METHOD BrakeStatus 								: REFERENCE TO Tc2_MC2.ST_McOutputs
VAR_INPUT
	bExecute									: BOOL;
END_VAR
VAR_INST
	{attribute 'hide'}
	fbRead										: Tc2_EtherCAT.FB_CoERead_ByDriveRef;
	{attribute 'hide'}
	ftRead										: F_TRIG;
	{attribute 'hide'}
	nData										: BYTE;
END_VAR
VAR
	Out											: Tc2_MC2.ST_McOutputs;
END_VAR
fbRead			(	stDriveRef				:= _stDriveRef, 
					nIndex					:= 16#3001 + (_stDriveRef.nDriveNo * 16#400), 
					nSubIndex				:= 16#07, 
					pDstBuf					:= ADR(nData), 
					cbBufLen				:= SIZEOF(nData), 
					bExecute				:= bExecute,
					bBusy					=> Out.Busy, 
					bError					=> Out.Error, 
					iAdsErrId				=> , 
					iCANopenErrId			=> );

IF Out.Error THEN
	Out.ErrorID								:= fbRead.iAdsErrId + fbRead.iCANopenErrId;
END_IF
					
ftRead(CLK:= Out.Busy, Q=> );
IF ftRead.Q THEN
	Out.Done								:= NOT Out.Error;
	bHoldingBrakeUnlocked					:= nData.0;
	bHoldingBrakeLocked						:= NOT nData.0;
END_IF

BrakeStatus									REF= Out;
END_METHOD

METHOD DeletePositionOffset 					: REFERENCE TO Tc2_MC2.ST_McOutputs
VAR_INPUT
	bExecute									: BOOL;
	eFeedback									: Tc2_MC2_Drive.E_PositionOffsetFeedback;
	eMemory										: Tc2_MC2_Drive.E_PositionOffsetMemory;
END_VAR
IF bExecute THEN
	DeletePositionOffsetEx(	eFeedback			:= eFeedback, 
							eMemory				:= eMemory);
ELSE
	DeletePositionOffsetClear();
END_IF

DeletePositionOffset							REF= pDeletePosOffs;
END_METHOD

METHOD DeletePositionOffsetClear 				: BOOL
VAR
	{attribute 'hide'}
	Out											: ST_McOutputs;
END_VAR
VAR_INST
	{attribute 'hide'}
	ftBusy										: F_TRIG;
END_VAR
fbDeletePositionOffset(	Axis					:= Axis, 
						Execute					:= FALSE, 
						Feedback				:= , 
						Memory					:= , 
						Busy					=> Out.Busy, 
						Error					=> Out.Error, 
						ErrorID					=> Out.ErrorID);

ftBusy(CLK:= Out.Busy, Q=> );						
IF ftBusy.Q THEN
	Out.Done									:= NOT Out.Error;
END_IF

pDeletePosOffs									REF= Out;

DeletePositionOffsetClear						:= TRUE;
END_METHOD

METHOD DeletePositionOffsetEncoder 				: REFERENCE TO Tc2_MC2.ST_McOutputs
VAR_INPUT
	bExecute									: BOOL;
END_VAR
DeletePositionOffset(	bExecute				:= bExecute,
						eFeedback				:= Tc2_MC2_Drive.E_PositionOffsetFeedback.ePositionOffsetFeedback1, 
						eMemory					:= Tc2_MC2_Drive.E_PositionOffsetMemory.ePositionOffsetMemory_Encoder);

DeletePositionOffsetEncoder						REF= pDeletePosOffs;
END_METHOD

METHOD DeletePositionOffsetEx 					: BOOL
VAR_INPUT
	eFeedback									: Tc2_MC2_Drive.E_PositionOffsetFeedback;
	eMemory										: Tc2_MC2_Drive.E_PositionOffsetMemory;
END_VAR
VAR
	{attribute 'hide'}
	Out											: ST_McOutputs;
END_VAR
fbDeletePositionOffset(	Axis					:= Axis, 
						Execute					:= TRUE, 
						Feedback				:= eFeedback, 
						Memory					:= eMemory, 
						Busy					=> Out.Busy, 
						Error					=> Out.Error, 
						ErrorID					=> Out.ErrorID);
						
Out.Done										:= NOT Out.Error AND NOT Out.Busy;
pDeletePosOffs									REF= Out;

DeletePositionOffsetEx							:= TRUE;
END_METHOD

METHOD FB_Init 									: BOOL
VAR_INPUT
	bInitRetains 								: BOOL; // if TRUE, the retain variables are initialized (warm start / cold start)
	bInCopyCode 								: BOOL;  // if TRUE, the instance afterwards gets moved into the copy code (online change)
END_VAR
pDeletePosOffs									REF= _stDeletePosOffs;
pSetPosOffs										REF= _stSetPosOffs;
pDriveAddress									REF= _stDriveAddress;
pDriveRef										REF= _stDriveRef;
END_METHOD

{attribute 'monitoring' := 'variable'}
PROPERTY fTorqueLimit 					: LREAL
GET
fTorqueLimit									:= nBipolarTorqueLimitValue/10.0;
END_GET
SET
VAR CONSTANT
	rTorqueLimitLow								: REAL 		:= 0.01;				// Low limit used for bipolar torque limit value
	rTorqueLimitHigh							: REAL		:= 500.0;				// High limit used for bipolar torque limit value
END_VAR
IF fTorqueLimit < rTorqueLimitLow OR fTorqueLimit > rTorqueLimitHigh THEN
	nBipolarTorqueLimitValue 					:= LREAL_TO_UINT(rTorqueLimitHigh)*10;
ELSE
	nBipolarTorqueLimitValue 					:= LREAL_TO_UINT(fTorqueLimit)*10;
END_IF
END_SET
END_PROPERTY

METHOD PRIVATE GetDriveRef 						: REFERENCE TO Tc2_MC2.ST_McOutputs
VAR_INPUT
	bExecute									: BOOL;
END_VAR
VAR_INST
	{attribute 'hide'}
	fbGetDriveRef								: FB_GetDriveRef;
	{attribute 'hide'}
	ftRead										: F_TRIG;
END_VAR
VAR
	{attribute 'hide'}
	Out											: Tc2_MC2.ST_McOutputs;
END_VAR
fbGetDriveRef(	bExecute						:= bExecute, 
				bBusy							=> Out.Busy, 
				bError							=> Out.Error, 
				udiErrorID						=> Out.ErrorID, 
				stDriveRef						=> _stDriveRef, 
				Axis							:= Axis);
				
ftRead(CLK:= Out.Busy, Q=> );
IF ftRead.Q THEN
	Out.Done									:= NOT Out.Error;
END_IF

GetDriveRef										REF= Out;
END_METHOD

METHOD HomingTorqueEncMemory 					: REFERENCE TO Tc2_MC2.ST_McOutputs
VAR_INPUT
	bExecute									: BOOL;					// The command is executed with a rising edge.
	fSetPos										: LREAL;
	bLagBased									: BOOL;					// TRUE: MC_StepBlockLagBased, FALSE: MC_StepBlock
	eDirection									: Tc3_MC2_AdvancedHoming.MC_Home_Direction;	// 
	fVelocity									: LREAL;				// Maximum travel velocity (>0)
	fDetectionVelocityLimit						: LREAL;				// Velocity that must be fallen below for the time DetectionVelocityTime in order to detect driving against the fixed stop.
	tDetectionVelocityTime						: TIME;					// Time for detecting the velocity undershoot when driving against the fixed stop.
	tTimeLimit									: TIME;					// Exceeding this time leads to the search procedure being aborted.
	fDistanceLimit								: LREAL;				// Exceeding this distance in relation to the start position leads to the search procedure being aborted.
	fTorqueLimit								: LREAL;				// The motor torque is limited to this value, in relation to the weight counterbalance that is possibly parameterized in the drive, in order to avoid mechanical damage.
	fTorqueTolerance							: LREAL;				// Tolerance related to the TorqueLimit within which driving against the fixed stop is detected.
	fLagLimit									: LREAL;				// Position lag value which, if exceeded, leads to detection of driving against the fixed stop.
	fDistance									: LREAL;				// Distance by which the axis moves away from the current position.
END_VAR
VAR_INST
	{attribute 'hide'}
	fbHomingTorque								: FB_HomingTorqueDetection;
	{attribute 'hide'}
	nStep										: DINT;
	{attribute 'hide'}
	fRecordedPosition							: LREAL;
	{attribute 'hide'}
	tonDelay									: TON;
	{attribute 'hide'}
	fSetPos_m									: LREAL;
END_VAR
VAR
	{attribute 'hide'}
	Out											: Tc2_MC2.ST_McOutputs;
	{attribute 'hide'}
	_HomingTorqueEncMemory						: Tc2_MC2.ST_McOutputs;
END_VAR
CASE nStep OF
	
	0: 
	
		IF bExecute THEN
			
			fbHomingTorque(	
				Axis							:= Axis, 
				bExecute						:= TRUE, 
				bLagBased						:= bLagBased, 
				eDirection						:= eDirection, 
				fVelocity						:= fVelocity, 
				fDetectionVelocityLimit			:= fDetectionVelocityLimit, 
				tDetectionVelocityTime			:= tDetectionVelocityTime, 
				tTimeLimit						:= tTimeLimit, 
				fDistanceLimit					:= fDistanceLimit, 
				fTorqueLimit					:= fTorqueLimit, 
				fTorqueTolerance				:= fTorqueTolerance, 
				fLagLimit						:= fLagLimit, 
				fDistance						:= fDistance);
				
			fSetPos_m							:= fSetPos;
		
			nStep								:= nStep + 10;
		
		END_IF
		
	10:
	
		fbHomingTorque(Axis := Axis);
		IF fbHomingTorque.bDone THEN
			fRecordedPosition 					:= fbHomingTorque.fRecordedPosition;
			fbHomingTorque(Axis := Axis, bExecute := FALSE);
			nStep								:= nStep + 10;
		ELSIF fbHomingTorque.bError OR fbHomingTorque.bCommandAborted THEN
			fbHomingTorque(Axis := Axis, bExecute := FALSE);
			nStep								:= nStep + 10_000;
		END_IF
		
	20:
	
		IF bHoldingBrakePresent THEN
			nStep								:= nStep + 10;
		ELSE
			nStep								:= 100;			
		END_IF
	
	30:
	
		Out 									:= BrakeForceLock();
		IF Out.Done THEN
			nStep								:= nStep + 10;
		ELSIF Out.Error OR Out.CommandAborted THEN
			nStep								:= nStep + 10_000;
		END_IF
		
	40:
	
		tonDelay(IN:= TRUE, PT:= T#1S);
		IF tonDelay.Q THEN
			tonDelay(IN:= FALSE);
			nStep								:= nStep + 10;
		END_IF
		
	50:
	
		Out 									:= BrakeStatus(bExecute := TRUE);
		IF Out.Done THEN
			BrakeStatus(bExecute := FALSE);
			nStep								:= nStep + 10;
		ELSIF Out.Error OR Out.CommandAborted THEN
			BrakeStatus(bExecute := FALSE);
			nStep								:= nStep + 10_000;
		END_IF
		
	60:
	
		IF bHoldingBrakeLocked THEN
			nStep								:= 100;	
		ELSE
			nStep								:= nStep + 10_000;
		END_IF
		
	100:

		_bWritingEncoderOffset					:= TRUE;		// if forses MC_Power disable
		nStep									:= nStep + 10;
		
	110:
	
		tonDelay(IN:= TRUE, PT:= T#1S);
		IF NOT pPower.Done THEN
			tonDelay(IN:= FALSE);
			nStep								:= nStep + 10;
		ELSIF tonDelay.Q THEN
			tonDelay(IN:= FALSE);
			nStep								:= nStep + 10_000;
		END_IF
		
	120:
	
		Out := SetPositionOffsetEncoderAbs(bExecute := TRUE, fPosition := Axis.NcToPlc.ActPos - fRecordedPosition + fSetPos_m);
		IF Out.Done THEN
			_bWritingEncoderOffset				:= FALSE;
			SetPositionOffsetEncoderAbs(bExecute := FALSE, fPosition := Axis.NcToPlc.ActPos - fRecordedPosition + fSetPos_m);
			nStep								:= nStep + 10;
		ELSIF Out.Error OR Out.CommandAborted THEN
			_bWritingEncoderOffset				:= FALSE;
			SetPositionOffsetEncoderAbs(bExecute := FALSE, fPosition := Axis.NcToPlc.ActPos - fRecordedPosition + fSetPos_m);
			nStep								:= nStep + 10_000;
		END_IF
		
	130:
			
		tonDelay(IN:= TRUE, PT:= T#1S);
		IF pPower.Done THEN
			tonDelay(IN:= FALSE);
			nStep								:= nStep + 10;
		ELSIF tonDelay.Q THEN
			tonDelay(IN:= FALSE);
			nStep								:= nStep + 10_000;
		END_IF
		
	140:
	
		IF bHoldingBrakePresent THEN
			nStep								:= nStep + 10;
		ELSE
			nStep								:= 1000;			
		END_IF
	
	150:
	
		Out 									:= BrakeReleaseForce();
		IF Out.Done THEN
			nStep								:= nStep + 10;
		ELSIF Out.Error OR Out.CommandAborted THEN
			nStep								:= nStep + 10_000;
		END_IF
		
	160:
	
		tonDelay(IN:= TRUE, PT:= T#1S);
		IF tonDelay.Q THEN
			tonDelay(IN:= FALSE);
			nStep								:= nStep + 10;
		END_IF
		
	170:
	
		Out 									:= BrakeStatus(bExecute := TRUE);
		IF Out.Done THEN
			BrakeStatus(bExecute := FALSE);
			nStep								:= nStep + 10;
		ELSIF Out.Error OR Out.CommandAborted THEN
			BrakeStatus(bExecute := FALSE);
			nStep								:= nStep + 10_000;
		END_IF
		
	180:
	
		IF bHoldingBrakeUnlocked THEN
			nStep								:= 1000;
		ELSE
			nStep								:= nStep + 10_000;
		END_IF
			
	1000:
		
		_HomingTorqueEncMemory.Done				:= TRUE;
		IF NOT bExecute THEN
			nStep 								:= 0;
		END_IF
		
	10_000..20_000:
	
		Out 									:= BrakeReleaseForce();
		_bWritingEncoderOffset					:= FALSE;
		IF NOT Out.Busy THEN
			nStep								:= 20_001;
		END_IF
		
	20_001:
	
		IF NOT bExecute THEN
			nStep 								:= 0;
		END_IF	
		
END_CASE

// States
_HomingTorqueEncMemory.Busy						:= (nStep > 0 AND nStep <= 1000) AND NOT _HomingTorqueEncMemory.Done;
_HomingTorqueEncMemory.Error					:= nStep >= 10_000;

HomingTorqueEncMemory							REF= _HomingTorqueEncMemory;
END_METHOD

METHOD PROTECTED Init 							: BOOL
VAR_INPUT
END_VAR
VAR_INST
	{attribute 'hide'}
	nStep										: DINT;
END_VAR
VAR
	{attribute 'hide'}
	Out											: ST_McOutputs;
	{attribute 'hide'}
	bNC_Initialized								: BOOL;
END_VAR
bNC_Initialized := SUPER^.Init();

CASE nStep OF
	
	0:	// Init
	
		IF bNC_Initialized THEN
			nStep								:= nStep + 10;
		END_IF

	10: // 

		Out := ReadDriveAddress(bExecute := TRUE);
		nStep									:= nStep + 10;

	20: //

		Out := ReadDriveAddress(bExecute := TRUE);
		IF Out.Done THEN
			Out := ReadDriveAddress(bExecute := FALSE);
			nStep								:= nStep + 10;
		ELSIF Out.Error THEN
			Out := ReadDriveAddress(bExecute := FALSE);
			nStep								:= nStep - 10;
		END_IF
		
	30: // 

		Out := GetDriveRef(bExecute := TRUE);
		nStep									:= nStep + 10;

	40: //

		Out := GetDriveRef(bExecute := TRUE);
		IF Out.Done THEN
			Out := GetDriveRef(bExecute := FALSE);
			nStep								:= nStep + 10;
		ELSIF Out.Error THEN
			Out := GetDriveRef(bExecute := FALSE);
			nStep								:= nStep - 10;
		END_IF
		
	50:
	
		Out := BrakePresent(bExecute := TRUE);
		nStep									:= nStep + 10;		

	60: //

		Out := BrakePresent(bExecute := TRUE);
		IF Out.Done THEN
			Out := BrakePresent(bExecute := FALSE);
			nStep								:= 100;
		ELSIF Out.Error THEN
			Out := BrakePresent(bExecute := FALSE);
			nStep								:= nStep - 10;
		END_IF
		
	100:
	
		Init									:= TRUE;

		IF NOT bNC_Initialized THEN
			nStep 								:= 0;
		END_IF

END_CASE
END_METHOD

{attribute 'monitoring' := 'variable'}
PROPERTY pDeletePosOffs 						: REFERENCE TO Tc2_MC2.ST_McOutputs
GET
pDeletePosOffs									REF= _stDeletePosOffs;
END_GET
SET
_stDeletePosOffs								:= pDeletePosOffs;
END_SET
END_PROPERTY

{attribute 'monitoring' := 'variable'}
PROPERTY pDriveAddress 							: REFERENCE TO Tc2_MC2.ST_DriveAddress
GET
pDriveAddress									REF= _stDriveAddress;
END_GET
SET
_stDriveAddress									:= pDriveAddress;
END_SET
END_PROPERTY

{attribute 'monitoring' := 'variable'}
PROPERTY pDriveRef 								: REFERENCE TO Tc2_EtherCAT.ST_DriveRef
GET
pDriveRef										REF= _stDriveRef;
END_GET
SET
_stDriveRef										:= pDriveRef;
END_SET
END_PROPERTY

METHOD Power 									: REFERENCE TO Tc2_MC2.ST_McOutputs
// SS1 read status and STO from AX8000

IF bEnable AND NOT pEStop.Done AND nSafetyState.0 AND NOT _bWritingEncoderOffset THEN
	Enable();
ELSE
	Disable();
END_IF

Power											REF= pPower;
END_METHOD

{attribute 'monitoring' := 'variable'}
PROPERTY pSetPosOffs 							: REFERENCE TO Tc2_MC2.ST_McOutputs
GET
pSetPosOffs										:= _stSetPosOffs;
END_GET
SET
_stSetPosOffs									:= pSetPosOffs;
END_SET
END_PROPERTY

METHOD PRIVATE ReadDriveAddress 				: REFERENCE TO Tc2_MC2.ST_McOutputs
VAR_INPUT
	bExecute									: BOOL;
END_VAR
VAR_INST
	{attribute 'hide'}
	mcReadDriveAddress							: Tc2_MC2.MC_ReadDriveAddress;
END_VAR
VAR
	{attribute 'hide'}
	Out											: Tc2_MC2.ST_McOutputs;
END_VAR
mcReadDriveAddress(	Axis						:= Axis,
					Execute						:= bExecute,
					Done						=> Out.Done,
					Busy						=> Out.Busy,
					Error						=> Out.Error,
					ErrorID						=> Out.ErrorID,
					DriveAddress				=> _stDriveAddress);

ReadDriveAddress								REF= Out;
END_METHOD

METHOD ReadI2T 							: BOOL
;
END_METHOD

METHOD ReadMotionPowerData 						: BOOL
;
END_METHOD

// very beta version
METHOD ReadMotorTorque 							: LREAL
ReadMotorTorque									:= Axis.NcToPlc.ActTorque;
END_METHOD

METHOD SetPositionOffset 						: REFERENCE TO Tc2_MC2.ST_McOutputs
VAR_INPUT
	bExecute									: BOOL;
	fPosition									: LREAL;
	bRelative									: BOOL;
	eFeedback									: Tc2_MC2_Drive.E_PositionOffsetFeedback;
	eMemory										: Tc2_MC2_Drive.E_PositionOffsetMemory;
END_VAR
IF bExecute THEN
	SetPositionOffsetEx(	fPosition			:= fPosition, 
							bRelative			:= bRelative, 
							eFeedback			:= eFeedback, 
							eMemory				:= eMemory);
ELSE
	SetPositionOffsetClear();
END_IF

SetPositionOffset								REF= pSetPosOffs;
END_METHOD

METHOD SetPositionOffsetClear 					: BOOL
VAR
	{attribute 'hide'}
	Out											: ST_McOutputs;
END_VAR
VAR_INST
	{attribute 'hide'}
	ftBusy										: F_TRIG;
END_VAR
fbSetPositionOffset(	Axis					:= Axis, 
						Execute					:= FALSE, 
						Position				:= , 
						Relative				:= , 
						Feedback				:= , 
						Memory					:= , 
						Busy					=> Out.Busy, 
						Error					=> Out.Error, 
						ErrorID					=> Out.ErrorID);

ftBusy(CLK:= Out.Busy, Q=> );						
IF ftBusy.Q THEN
	Out.Done									:= NOT Out.Error;
END_IF

pSetPosOffs										REF= Out;

SetPositionOffsetClear							:= TRUE;
END_METHOD

METHOD SetPositionOffsetEncoderAbs 				: REFERENCE TO Tc2_MC2.ST_McOutputs
VAR_INPUT
	bExecute									: BOOL;
	fPosition									: LREAL;
END_VAR
SetPositionOffset(		bExecute				:= bExecute, 
						fPosition				:= fPosition, 
						bRelative				:= FALSE, 
						eFeedback				:= Tc2_MC2_Drive.E_PositionOffsetFeedback.ePositionOffsetFeedback1, 
						eMemory					:= Tc2_MC2_Drive.E_PositionOffsetMemory.ePositionOffsetMemory_Encoder);

SetPositionOffsetEncoderAbs						REF= pSetPosOffs;
END_METHOD

METHOD SetPositionOffsetEncoderAbsZero 			: REFERENCE TO Tc2_MC2.ST_McOutputs
VAR_INPUT
	bExecute									: BOOL;
END_VAR
SetPositionOffset(		bExecute				:= bExecute, 
						fPosition				:= 0.0, 
						bRelative				:= FALSE, 
						eFeedback				:= Tc2_MC2_Drive.E_PositionOffsetFeedback.ePositionOffsetFeedback1, 
						eMemory					:= Tc2_MC2_Drive.E_PositionOffsetMemory.ePositionOffsetMemory_Encoder);

SetPositionOffsetEncoderAbsZero					REF= pSetPosOffs;
END_METHOD

METHOD SetPositionOffsetEncoderRel 				: REFERENCE TO Tc2_MC2.ST_McOutputs
VAR_INPUT
	bExecute									: BOOL;
	fPosition									: LREAL;
END_VAR
SetPositionOffset(		bExecute				:= bExecute, 
						fPosition				:= fPosition, 
						bRelative				:= TRUE, 
						eFeedback				:= Tc2_MC2_Drive.E_PositionOffsetFeedback.ePositionOffsetFeedback1, 
						eMemory					:= Tc2_MC2_Drive.E_PositionOffsetMemory.ePositionOffsetMemory_Encoder);

SetPositionOffsetEncoderRel						REF= pSetPosOffs;
END_METHOD

METHOD SetPositionOffsetEx 						: BOOL
VAR_INPUT
	fPosition									: LREAL;
	bRelative									: BOOL;
	eFeedback									: Tc2_MC2_Drive.E_PositionOffsetFeedback;
	eMemory										: Tc2_MC2_Drive.E_PositionOffsetMemory;
END_VAR
VAR
	{attribute 'hide'}
	Out											: ST_McOutputs;
END_VAR
fbSetPositionOffset(	Axis					:= Axis, 
						Execute					:= TRUE, 
						Position				:= fPosition, 
						Relative				:= bRelative, 
						Feedback				:= eFeedback, 
						Memory					:= eMemory, 
						Busy					=> Out.Busy, 
						Error					=> Out.Error, 
						ErrorID					=> Out.ErrorID);
						
Out.Done										:= NOT Out.Error AND NOT Out.Busy;
pSetPosOffs										REF= Out;

SetPositionOffsetEx								:= TRUE;
END_METHOD

METHOD TorqueControl 							: REFERENCE TO Tc2_MC2.ST_McOutputs
VAR_INPUT
	bExecute									: BOOL;
END_VAR
END_METHOD

METHOD TorqueControlClear 						: BOOL
END_METHOD

METHOD TorqueControlEx 							: BOOL
END_METHOD

END_FUNCTION_BLOCK

// ---- POUs/FB/AxisControl/Base/FB_AxisBase.TcPOU
//==================================================================================================
//							Beckhoff Automation Poland
//									03.01.2023
//
// Code owner: TG
//
// Sample code to handle NC Axis
//
// Used libraries: 
//	Tc2_MC2								|| 3.3.48.0
//	Tc2_System							|| 3.4.26.0
//
// Used DUTs:
//	ST_AxisControlManual
//
// Used FBs:
//	FB_NcSWLimitSwitchCtrl
//
//  v1.0	|| TC v 3.1.4024.35		|| First edition
//==================================================================================================
{attribute 'reflection'}
FUNCTION_BLOCK FB_AxisBase IMPLEMENTS I_AxisControlBase
VAR	
	Axis										: Tc2_MC2.AXIS_REF;
	{attribute 'instance-path'}
	{attribute 'noinit'}
	sInstancePath								: STRING;
	stParameters								: Tc2_MC2.ST_AxisParameterSet;
	// Manual Motion
	stManualHMI									: ST_AxisControlManualHMI;	// Base manual motion + base HMI handling
	// Flags
	bAxisRefError								: BOOL;
	bMasterAxisRefError							: BOOL;
	// Properties
	{attribute 'hide'}
	_bEnable									: BOOL;
	{attribute 'hide'}
	_bEnablePositive							: BOOL;
	{attribute 'hide'}
	_bEnableNegative							: BOOL;
	{attribute 'hide'}
	_bExecuteEstop								: BOOL;							// Executes SS1 cmd	
	{attribute 'hide'}
	_fOverride									: LREAL;
	{attribute 'hide'}
	_fAcceleration								: LREAL 		:= 0.0;
	{attribute 'hide'}
	_fDeceleration								: LREAL 		:= 0.0;
	{attribute 'hide'}
	_fJerk										: LREAL 		:= 0.0;
	{attribute 'hide'}
	_fDecelerationEstop							: LREAL 		:= 0.0;
	{attribute 'hide'}
	_fJerkEstop									: LREAL 		:= 0.0;
	{attribute 'hide'}
	_fPosition									: LREAL 		:= 0.0;
	{attribute 'hide'}
	_fDistance									: LREAL 		:= 0.0;
	{attribute 'hide'}
	_fVelocity									: LREAL 		:= 0.0;
	{attribute 'hide'}
	_fGearRatio									: LREAL 		:= 0.0;
	{attribute 'hide'}
	_fLimitSwitchPositionMin					: LREAL 		:= 0.0;
	{attribute 'hide'}
	_fLimitSwitchPositionMax					: LREAL 		:= 0.0;
	{attribute 'hide'}
	_bLimitSwitchStateMin						: BOOL 			:= FALSE;
	{attribute 'hide'}
	_bLimitSwitchStateMax						: BOOL 			:= FALSE;
	
	{attribute 'hide'}
	_eDirection									: Tc2_MC2.MC_Direction;
	{attribute 'hide'}
	_eBufferMode								: Tc2_MC2.MC_BufferMode;
	{attribute 'hide'}
	_eJogMode									: Tc2_MC2.E_JogMode;
	
	// FBs
	{attribute 'hide'}
	_stOut										: Tc2_MC2.ST_McOutputs;
	{attribute 'hide'}
	mcPower										: Tc2_MC2.MC_Power;
	{attribute 'hide'}
	_stPower									: Tc2_MC2.ST_McOutputs;
	{attribute 'hide'}
	mcReset										: Tc2_MC2.MC_Reset;
	{attribute 'hide'}
	_stReset									: Tc2_MC2.ST_McOutputs;
	{attribute 'hide'}
	mcSetPos									: Tc2_MC2.MC_SetPosition;
	{attribute 'hide'}
	_stSetPos									: Tc2_MC2.ST_McOutputs;
	{attribute 'hide'}
	mcMoveAbsolute								: Tc2_MC2.MC_MoveAbsolute;
	{attribute 'hide'}
	_stAbsolute									: Tc2_MC2.ST_McOutputs;
	{attribute 'hide'}
	mcMoveAbsolute2								: Tc2_MC2.MC_MoveAbsolute;
	{attribute 'hide'}
	_stAbsolute2								: Tc2_MC2.ST_McOutputs;
	{attribute 'hide'}
	mcEStop										: Tc2_MC2.MC_Stop;
	{attribute 'hide'}
	_stEStop									: Tc2_MC2.ST_McOutputs;
	{attribute 'hide'}
	mcStop										: Tc2_MC2.MC_Stop;
	{attribute 'hide'}
	_stStop										: Tc2_MC2.ST_McOutputs;
	{attribute 'hide'}
	mcHalt										: Tc2_MC2.MC_Halt;
	{attribute 'hide'}
	_stHalt										: Tc2_MC2.ST_McOutputs;
	{attribute 'hide'}
	mcMoveRelative								: Tc2_MC2.MC_MoveRelative;
	{attribute 'hide'}
	_stRelative									: Tc2_MC2.ST_McOutputs;
	{attribute 'hide'}
	mcMoveRelative2								: Tc2_MC2.MC_MoveRelative;
	{attribute 'hide'}
	_stRelative2								: Tc2_MC2.ST_McOutputs;
	{attribute 'hide'}
	mcMoveVelocity								: Tc2_MC2.MC_MoveVelocity;
	{attribute 'hide'}
	_stVelocity									: Tc2_MC2.ST_McOutputs;
	{attribute 'hide'}
	mcMoveVelocity2								: Tc2_MC2.MC_MoveVelocity;
	{attribute 'hide'}
	_stVelocity2								: Tc2_MC2.ST_McOutputs;
	{attribute 'hide'}
	mcMoveModulo								: Tc2_MC2.MC_MoveModulo;
	{attribute 'hide'}
	_stModulo									: Tc2_MC2.ST_McOutputs;
	{attribute 'hide'}
	mcMoveModulo2								: Tc2_MC2.MC_MoveModulo;
	{attribute 'hide'}
	_stModulo2									: Tc2_MC2.ST_McOutputs;
	{attribute 'hide'}
	mcJog										: Tc2_MC2.MC_Jog;
	{attribute 'hide'}
	_stJog										: Tc2_MC2.ST_McOutputs;
	{attribute 'hide'}
	mcHome										: Tc2_MC2.MC_Home;
	{attribute 'hide'}
	_stHome										: Tc2_MC2.ST_McOutputs;
	{attribute 'hide'}
	mcGearIn									: Tc2_MC2.MC_GearIn;
	{attribute 'hide'}
	mcGearInDyn									: Tc2_MC2.MC_GearInDyn;
	{attribute 'hide'}
	mcGearInMulti								: Tc2_MC2.MC_GearInMultiMaster;
	{attribute 'hide'}
	mcGearOut									: Tc2_MC2.MC_GearOut;
	{attribute 'hide'}
	_stGear										: Tc2_MC2.ST_McOutputs;
	{attribute 'hide'}
	fbLimitSwitch								: FB_NcSWLimitSwitchCtrlv2;
	{attribute 'hide'}
	_stLimitSwitch								: Tc2_MC2.ST_McOutputs;
	{attribute 'hide'}
	fbPosLagMonitoring							: FB_NcPosLagMonitoring;
	
	mcMoveSuperimposed							: Tc2_MC2.MC_MoveSuperImposed;
	{attribute 'hide'}
	_stSuperimposed								: Tc2_MC2.ST_McOutputs;
		

END_VAR

Cyclic();

{attribute 'monitoring' := 'variable'}
PROPERTY bConsequentialError 					: BOOL
GET
bConsequentialError								:= IsConsequentialError(Axis.NcToPlc.ErrorCode);
END_GET
END_PROPERTY

{attribute 'monitoring' := 'variable'}
PROPERTY bDisabled 								: BOOL
GET
bDisabled										:= NOT bEnabled;
END_GET
END_PROPERTY

{attribute 'monitoring' := 'variable'}
PROPERTY bDriveError 							: BOOL
GET
bDriveError										:= Axis.Status.DriveDeviceError;
END_GET
END_PROPERTY

{attribute 'monitoring' := 'variable'}
PROPERTY bEnable 								: BOOL
GET
bEnable 										:= _bEnable;
END_GET
SET
_bEnable 										:= bEnable;
END_SET
END_PROPERTY

{attribute 'monitoring' := 'variable'}
PROPERTY bEnabled 								: BOOL
GET
bEnabled											:= Axis.Status.ControlLoopClosed;
END_GET
END_PROPERTY

{attribute 'monitoring' := 'variable'}
PROPERTY bEnableNegative 						: BOOL
GET
bEnableNegative 									:= _bEnableNegative;
END_GET
SET
_bEnableNegative 								:= bEnableNegative;
END_SET
END_PROPERTY

{attribute 'monitoring' := 'variable'}
PROPERTY bEnablePositive 						: BOOL
GET
bEnablePositive 									:= _bEnablePositive;
END_GET
SET
_bEnablePositive 								:= bEnablePositive;
END_SET
END_PROPERTY

{attribute 'monitoring' := 'variable'}
PROPERTY bError 									: BOOL
GET
bError											:= Axis.Status.Error;
END_GET
END_PROPERTY

{attribute 'monitoring' := 'variable'}
PROPERTY bErrorFB 							: BOOL
GET
bErrorFB										:= NOT bError AND
													(pPower.Error 
													OR pAbsolute.Error 
													OR pAbsolute2.Error 
													OR pEStop.Error 
													OR pGear.Error 
													OR pHalt.Error
													OR pHome.Error
													OR pJog.Error
													OR pModulo.Error
													OR pModulo2.Error
													OR pRelative.Error
													OR pRelative2.Error
													OR pReset.Error
													OR pSetPos.Error
													OR pStop.Error
													OR pSuperimposed.Error
													OR pVelocity.Error
													OR pVelocity2.Error);
END_GET
END_PROPERTY

{attribute 'monitoring' := 'variable'}
PROPERTY bErrorFiltered 									: BOOL
GET
bErrorFiltered									:= Axis.Status.Error AND NOT bConsequentialError;
END_GET
END_PROPERTY

{attribute 'monitoring' := 'variable'}
PROPERTY bExecuteEstop 							: BOOL
GET
bExecuteEstop 									:= _bExecuteEstop;
END_GET
SET
_bExecuteEstop 									:= bExecuteEstop;
END_SET
END_PROPERTY

{attribute 'monitoring' := 'variable'}
PROPERTY bExist 								: BOOL
GET
bExist											:= Axis.NcToPlc.AxisId <> 0;
END_GET
END_PROPERTY

{attribute 'monitoring' := 'variable'}
PROPERTY bHomed 								: BOOL
GET
bHomed											:= Axis.Status.Homed;
END_GET
END_PROPERTY

PROPERTY bLimitSwitchStateMax 					: BOOL
GET
bLimitSwitchStateMax								:= _bLimitSwitchStateMax;
END_GET
SET
_bLimitSwitchStateMax							:= bLimitSwitchStateMax;
END_SET
END_PROPERTY

PROPERTY bLimitSwitchStateMin 					: BOOL
GET
bLimitSwitchStateMin							:= _bLimitSwitchStateMin;
END_GET
SET
_bLimitSwitchStateMin							:= bLimitSwitchStateMin;
END_SET
END_PROPERTY

{attribute 'monitoring' := 'variable'}
PROPERTY bMoving 								: BOOL
GET
bMoving											:= Axis.Status.Moving;
END_GET
END_PROPERTY

{attribute 'monitoring' := 'variable'}
PROPERTY bNotMoving 								: BOOL
GET
bNotMoving										:= Axis.Status.NotMoving;
END_GET
END_PROPERTY

{attribute 'monitoring' := 'variable'}
PROPERTY bSimulationAxis 						: BOOL
GET
bSimulationAxis									:= Axis.Status.OpMode.SimulationAxis;
END_GET
END_PROPERTY

METHOD CheckAxisRef 							: BOOL
;
(*IF NOT __ISVALIDREF(Axis) THEN

	IF NOT bAxisRefError THEN
		ADSLOGSTR(ADSLOG_MSGTYPE_ERROR,'FB_AxisBase critical error - Axis Reference not assigned! FB instance: %s',sInstancePath);
	END_IF

	bAxisRefError 								:= TRUE;
	
	RETURN;

END_IF
*)
END_METHOD

METHOD ClearAll 								: BOOL
MoveAbsoluteClear();
MoveAbsoluteClear2();
MoveRelativeClear();
MoveRelativeClear2();
MoveVelocityClear();
MoveVelocityClear2();
MoveModuloClear();
MoveModuloClear2();

JogClear();
HomeClear(bCalibrationCam := FALSE);

HaltClear();
StopClear();

ResetClear();
SetPosClear();
END_METHOD

METHOD PRIVATE Cyclic 							: BOOL
Axis();
Axis.ReadStatus();
Init();
EStop(bExecute := bExecuteEstop);
Power();
END_METHOD

METHOD Disable 									: BOOL
VAR
	{attribute 'hide'}
	Out											: Tc2_MC2.ST_McOutputs;
END_VAR
bEnable 										:= FALSE;

mcPower(			Axis						:= Axis, 
					Enable						:= FALSE, 
					Enable_Positive				:= FALSE, 
					Enable_Negative				:= FALSE, 
					Override					:= fOverride, 
					BufferMode					:= , 
					Options						:= , 
					Status						=> Out.Done, 
					Busy						=> Out.Busy, 
					Active						=> Out.Active, 
					Error						=> Out.Error, 
					ErrorID						=> Out.ErrorID);
	
pPower											REF= Out;

Disable											:= TRUE;
END_METHOD

{attribute 'monitoring' := 'variable'}
PROPERTY eBufferMode 							: Tc2_MC2.MC_BufferMode
GET
eBufferMode 										:= _eBufferMode;
END_GET
SET
_eBufferMode 									:= eBufferMode;
END_SET
END_PROPERTY

{attribute 'monitoring' := 'variable'}
PROPERTY eDirection 								: Tc2_MC2.MC_Direction
GET
_eDirection										:= _eDirection;
END_GET
SET
_eDirection										:= _eDirection;
END_SET
END_PROPERTY

{attribute 'monitoring' := 'variable'}
PROPERTY eJogMode 								: Tc2_MC2.E_JogMode
GET
eJogMode 										:= _eJogMode;
END_GET
SET
_eJogMode 										:= eJogMode;
END_SET
END_PROPERTY

METHOD Enable 									: BOOL
VAR
	{attribute 'hide'}
	Out											: Tc2_MC2.ST_McOutputs;
	{attribute 'hide'}
	EstopOut									: Tc2_MC2.ST_McOutputs;
END_VAR
bEnable 										:= TRUE;

mcPower(			Axis						:= Axis, 
					Enable						:= bEnable, 
					Enable_Positive				:= bEnablePositive, 
					Enable_Negative				:= bEnableNegative, 
					Override					:= fOverride, 
					BufferMode					:= , 
					Options						:= , 
					Status						=> Out.Done, 
					Busy						=> Out.Busy, 
					Active						=> Out.Active, 
					Error						=> Out.Error, 
					ErrorID						=> Out.ErrorID);
	
pPower											REF= Out;

Enable											:= TRUE;
END_METHOD

// Has own Dcc, Jerk properties
METHOD EStop 									: REFERENCE TO Tc2_MC2.ST_McOutputs
VAR_INPUT
	bExecute									: BOOL;
END_VAR
IF bExecute THEN
	EStopEx();
ELSE
	EStopClear();
END_IF

EStop											REF= pEStop;
END_METHOD

METHOD EStopClear 								: BOOL
VAR
	{attribute 'hide'}
	Out											: Tc2_MC2.ST_McOutputs;
END_VAR
mcEStop(			Axis						:= Axis, 
					Execute						:= FALSE, 
					Done						=> Out.Done, 
					Busy						=> Out.Busy, 
					Active						=> Out.Active, 
					CommandAborted				=> Out.CommandAborted, 
					Error						=> Out.Error, 
					ErrorID						=> Out.ErrorID);

pEStop				 							REF= Out;

EStopClear										:= TRUE;
END_METHOD

METHOD EStopEx 									: BOOL
VAR
	{attribute 'hide'}
	Out											: Tc2_MC2.ST_McOutputs;
END_VAR
mcEStop(			Axis						:= Axis, 
					Execute						:= TRUE, 
					Deceleration				:= fDecelerationEstop, 
					Jerk						:= fJerkEstop, 
					Options						:= , 
					Done						=> Out.Done, 
					Busy						=> Out.Busy, 
					Active						=> Out.Active, 
					CommandAborted				=> Out.CommandAborted, 
					Error						=> Out.Error, 
					ErrorID						=> Out.ErrorID);

pEStop				 							REF= Out;

EStopEx											:= TRUE;
END_METHOD

{attribute 'monitoring' := 'variable'}
PROPERTY fAcceleration 							: LREAL
GET
fAcceleration 									:= _fAcceleration;
END_GET
SET
_fAcceleration 								:= fAcceleration;
END_SET
END_PROPERTY

{attribute 'monitoring' := 'variable'}
PROPERTY fActAcc 								: LREAL
GET
fActAcc											:= Axis.NcToPlc.ActAcc;
END_GET
END_PROPERTY

{attribute 'monitoring' := 'variable'}
PROPERTY fActPos 								: LREAL
GET
fActPos											:= Axis.NcToPlc.ActPos;
END_GET
END_PROPERTY

{attribute 'monitoring' := 'variable'}
PROPERTY fActTorque 								: LREAL
GET
fActTorque										:= Axis.NcToPlc.ActTorque;
END_GET
END_PROPERTY

{attribute 'monitoring' := 'variable'}
PROPERTY fActVelo 								: LREAL
GET
fActVelo											:= Axis.NcToPlc.ActVelo;
END_GET
END_PROPERTY

METHOD FB_Init 									: BOOL
VAR_INPUT
	bInitRetains 								: BOOL; // if TRUE, the retain variables are initialized (warm start / cold start)
	bInCopyCode 								: BOOL;  // if TRUE, the instance afterwards gets moved into the copy code (online change)
END_VAR
stManualHMI.stParameters						REF= stParameters;
stManualHMI.stStatus							REF= Axis.Status;
bEnablePositive									:= TRUE;
bEnableNegative									:= TRUE;
fOverride										:= 100.0;
// Online view before call <Deference of invalid pointer>
pPower											REF= _stPower;
pReset											REF= _stReset;
pSetPos											REF= _stSetPos;
pEStop											REF= _stEStop;
pStop											REF= _stStop;
pHalt											REF= _stHalt;
pStop											REF= _stStop;
pGear											REF= _stGear;
pLimitSwitch									REF= _stLimitSwitch;

pVelocity										REF= _stVelocity;
pVelocity2										REF= _stVelocity2;
pAbsolute										REF= _stAbsolute;
pAbsolute2										REF= _stAbsolute2;
pRelative										REF= _stRelative;
pRelative2										REF= _stRelative2;
pModulo											REF= _stModulo;
pModulo2										REF= _stModulo2;
pJog											REF= _stJog;
pHome											REF= _stHome;

pOut											REF= _stOut;
END_METHOD

{attribute 'monitoring' := 'variable'}
PROPERTY fDeceleration 							: LREAL
GET
fDeceleration 									:= _fDeceleration;
END_GET
SET
_fDeceleration 								:= fDeceleration;
END_SET
END_PROPERTY

{attribute 'monitoring' := 'variable'}
PROPERTY fDecelerationEstop 						: LREAL
GET
fDecelerationEstop 								:= _fDecelerationEstop;
END_GET
SET
_fDecelerationEstop 							:= fDecelerationEstop;
END_SET
END_PROPERTY

{attribute 'monitoring' := 'variable'}
PROPERTY fDistance 								: LREAL
GET
fDistance 										:= _fDistance;
END_GET
SET
_fDistance 									:= fDistance;
END_SET
END_PROPERTY

{attribute 'monitoring' := 'variable'}
PROPERTY fGearRatio 								: LREAL
GET
fGearRatio 										:= _fGearRatio;
END_GET
SET
_fGearRatio 									:= fGearRatio;
END_SET
END_PROPERTY

METHOD FilterConsequentialError 				: UDINT
VAR CONSTANT
	// Filtered Errors
	nConsequentialError							: UDINT 	:= 16#42A0; (*Group/axis consequential error" Consequential error resulting from another causative error 
																		related to another axis within the group. 
																		Group/axis consequential errors can occur in relation to master/slave couplings or 
																		with multiple axis interpolating DXD groups. 
																		If, for instance, it is detected that the following error limit of a master axis has been exceeded, 
																		then this consequential error is assigned to all the other master axes and slave axes in this group.*)
END_VAR
VAR_INPUT
	nErrorID									: UDINT;
END_VAR
CASE nErrorID OF
	
	0, nConsequentialError:
	
		; // Do nothing
		
ELSE
	
	FilterConsequentialError					:= nErrorID;
	
END_CASE
END_METHOD

{attribute 'monitoring' := 'variable'}
PROPERTY fJerk 									: LREAL
GET
fJerk 											:= _fJerk;
END_GET
SET
_fJerk 										:= fJerk;
END_SET
END_PROPERTY

{attribute 'monitoring' := 'variable'}
PROPERTY fJerkEstop 								: LREAL
GET
fJerkEstop 										:= _fJerkEstop;
END_GET
SET
_fJerkEstop 									:= fJerkEstop;
END_SET
END_PROPERTY

PROPERTY fLimitSwitchPositionMax 				: LREAL
GET
fLimitSwitchPositionMax							:= _fLimitSwitchPositionMax;
END_GET
SET
_fLimitSwitchPositionMax						:= fLimitSwitchPositionMax;
END_SET
END_PROPERTY

PROPERTY fLimitSwitchPositionMin 				: LREAL
GET
fLimitSwitchPositionMin							:= _fLimitSwitchPositionMin;
END_GET
SET
_fLimitSwitchPositionMin						:= fLimitSwitchPositionMin;
END_SET
END_PROPERTY

{attribute 'monitoring' := 'variable'}
PROPERTY fOverride 								: LREAL
GET
fOverride 										:= _fOverride;
END_GET
SET
_fOverride 									:= fOverride;
END_SET
END_PROPERTY

{attribute 'monitoring' := 'variable'}
PROPERTY fPosition 								: LREAL
GET
fPosition 										:= _fPosition;
END_GET
SET
_fPosition 									:= fPosition;
END_SET
END_PROPERTY

{attribute 'monitoring' := 'variable'}
PROPERTY fSetAcc 								: LREAL
GET
fSetAcc											:= Axis.NcToPlc.SetAcc;
END_GET
END_PROPERTY

{attribute 'monitoring' := 'variable'}
PROPERTY fSetPos 								: LREAL
GET
fSetPos											:= Axis.NcToPlc.SetPos;
END_GET
END_PROPERTY

{attribute 'monitoring' := 'variable'}
PROPERTY fSetVelo 								: LREAL
GET
fSetVelo											:= Axis.NcToPlc.SetVelo;
END_GET
END_PROPERTY

{attribute 'monitoring' := 'variable'}
PROPERTY fVelocity 								: LREAL
GET
fVelocity 										:= _fVelocity;
END_GET
SET
_fVelocity 									:= fVelocity;
END_SET
END_PROPERTY

METHOD GearIn 									: REFERENCE TO Tc2_MC2.ST_McOutputs
VAR_INPUT
	bExecute									: BOOL;
	Master										: REFERENCE TO Tc2_MC2.AXIS_REF;
END_VAR
IF bExecute THEN
	GearInEx(Master := Master);
ELSE
	GearInClear(Master := Master);
END_IF

GearIn											REF= pGear;
END_METHOD

METHOD GearInClear 								: BOOL
VAR_INPUT
	Master										: REFERENCE TO Tc2_MC2.AXIS_REF;
END_VAR
VAR
	{attribute 'hide'}
	Out											: Tc2_MC2.ST_McOutputs;
END_VAR
IF NOT __ISVALIDREF(Master) THEN

	IF NOT bMasterAxisRefError THEN
		ADSLOGSTR(ADSLOG_MSGTYPE_ERROR,'FB_AxisBase critical error - Master Axis Reference not assigned! FB instance: %s',sInstancePath);
	END_IF

	bMasterAxisRefError 						:= TRUE;
	
	RETURN;

END_IF

mcGearIn(			Master						:= Master, 
					Slave						:= Axis, 
					Execute						:= FALSE,
					InGear						=> Out.Done, 
					Busy						=> Out.Busy, 
					Active						=> Out.Active, 
					CommandAborted				=> Out.CommandAborted, 
					Error						=> Out.Error, 
					ErrorID						=> Out.ErrorID);
					
pGear 											REF= Out;

GearInClear										:= TRUE;
END_METHOD

METHOD GearInDyn 								: REFERENCE TO Tc2_MC2.ST_McOutputs
VAR_INPUT
	bEnable										: BOOL;
	Master										: REFERENCE TO Tc2_MC2.AXIS_REF;
END_VAR
IF bEnable THEN
	GearInDynEx(Master := Master);
ELSE
	GearInDynClear(Master := Master);
END_IF

GearInDyn										REF= pGear;
END_METHOD

METHOD GearInDynClear 							: BOOL
VAR_INPUT
	Master										: REFERENCE TO Tc2_MC2.AXIS_REF;
END_VAR
VAR
	{attribute 'hide'}
	Out											: Tc2_MC2.ST_McOutputs;
END_VAR
//CheckAxisRef();

IF NOT __ISVALIDREF(Master) THEN

	IF NOT bMasterAxisRefError THEN
		ADSLOGSTR(ADSLOG_MSGTYPE_ERROR,'FB_AxisBase critical error - Master Axis Reference not assigned! FB instance: %s',sInstancePath);
	END_IF

	bMasterAxisRefError 						:= TRUE;
	
	RETURN;

END_IF

mcGearInDyn(		Master						:= Master, 
					Slave						:= Axis, 
					Enable						:= FALSE,
					InGear						=> Out.Done, 
					Busy						=> Out.Busy, 
					Active						=> Out.Active, 
					CommandAborted				=> Out.CommandAborted, 
					Error						=> Out.Error, 
					ErrorID						=> Out.ErrorID);
					
pGear 											REF= Out;

GearInDynClear									:= TRUE;
END_METHOD

METHOD GearInDynEq 								: REFERENCE TO Tc2_MC2.ST_McOutputs
VAR_INPUT
	bEnable										: BOOL;
	Master										: REFERENCE TO Tc2_MC2.AXIS_REF;
END_VAR
IF bEnable THEN
	fGearRatio 									:= 1.0;
	GearInDynEx(Master := Master);
ELSE
	GearInDynClear(Master := Master);
END_IF

GearInDynEq										REF= pGear;
END_METHOD

METHOD GearInDynEx 								: BOOL
VAR_INPUT
	Master										: REFERENCE TO Tc2_MC2.AXIS_REF;
END_VAR
VAR
	{attribute 'hide'}
	Out											: Tc2_MC2.ST_McOutputs;
END_VAR
IF NOT __ISVALIDREF(Master) THEN

	IF NOT bMasterAxisRefError THEN
		ADSLOGSTR(ADSLOG_MSGTYPE_ERROR,'FB_AxisBase critical error - Master Axis Reference not assigned! FB instance: %s',sInstancePath);
	END_IF

	bMasterAxisRefError 						:= TRUE;
	
	RETURN;

END_IF

mcGearInDyn(		Master						:= Master, 
					Slave						:= Axis, 
					Enable						:= TRUE, 
					GearRatio					:= fGearRatio, 
					InGear						=> Out.Done, 
					Busy						=> Out.Busy, 
					Active						=> Out.Active, 
					CommandAborted				=> Out.CommandAborted, 
					Error						=> Out.Error, 
					ErrorID						=> Out.ErrorID);
					
pGear 											REF= Out;

GearInDynEx										:= TRUE;
END_METHOD

METHOD GearInDynOpposite 						: REFERENCE TO Tc2_MC2.ST_McOutputs
VAR_INPUT
	bEnable										: BOOL;
	Master										: REFERENCE TO Tc2_MC2.AXIS_REF;
END_VAR
IF bEnable THEN
	fGearRatio 									:= -1.0;
	GearInDynEx(Master := Master);
ELSE
	GearInDynClear(Master := Master);
END_IF

GearInDynOpposite								REF= pGear;
END_METHOD

METHOD GearInEq 								: REFERENCE TO Tc2_MC2.ST_McOutputs
VAR_INPUT
	bExecute									: BOOL;
	Master										: REFERENCE TO Tc2_MC2.AXIS_REF;
END_VAR
IF bExecute THEN
	fGearRatio 									:= 1.0;
	GearInEx(Master := Master);
ELSE
	GearInClear(Master := Master);
END_IF

GearInEq										REF= pGear;
END_METHOD

METHOD GearInEx 								: BOOL
VAR_INPUT
	Master										: REFERENCE TO Tc2_MC2.AXIS_REF;
END_VAR
VAR
	{attribute 'hide'}
	Out											: Tc2_MC2.ST_McOutputs;
END_VAR
IF NOT __ISVALIDREF(Master) THEN

	IF NOT bMasterAxisRefError THEN
		ADSLOGSTR(ADSLOG_MSGTYPE_ERROR,'FB_AxisBase critical error - Master Axis Reference not assigned! FB instance: %s',sInstancePath);
	END_IF

	bMasterAxisRefError 						:= TRUE;
	
	RETURN;

END_IF

mcGearIn(			Master						:= Master, 
					Slave						:= Axis, 
					Execute						:= TRUE, 
					RatioNumerator				:= fGearRatio, 
					RatioDenominator			:= 1,
					InGear						=> Out.Done, 
					Busy						=> Out.Busy, 
					Active						=> Out.Active, 
					CommandAborted				=> Out.CommandAborted, 
					Error						=> Out.Error, 
					ErrorID						=> Out.ErrorID);
					
pGear 											REF= Out;

GearInEx										:= TRUE;
END_METHOD

METHOD GearInOpposite 							: REFERENCE TO Tc2_MC2.ST_McOutputs
VAR_INPUT
	bExecute									: BOOL;
	Master										: REFERENCE TO Tc2_MC2.AXIS_REF;
END_VAR
IF bExecute THEN
	fGearRatio 									:= -1.0;
	GearInEx(Master := Master);
ELSE
	GearInClear(Master := Master);
END_IF

GearInOpposite									REF= pGear;
END_METHOD

METHOD GearOut 									: REFERENCE TO Tc2_MC2.ST_McOutputs
VAR_INPUT
	bExecute									: BOOL;
END_VAR
IF bExecute THEN
	GearOutEx();
ELSE
	GearOutClear();
END_IF

GearOut											REF= pGear;
END_METHOD

METHOD GearOutClear 							: BOOL
VAR
	{attribute 'hide'}
	Out											: Tc2_MC2.ST_McOutputs;
END_VAR
mcGearOut( 			Slave						:= Axis, 
					Execute						:= FALSE, 
					Done						=> Out.Done, 
					Busy						=> Out.Busy, 
					Error						=> Out.Error, 
					ErrorID						=> Out.ErrorID);

					
pGear 											REF= Out;

GearOutClear									:= TRUE;
END_METHOD

METHOD GearOutEx 								: BOOL
VAR
	{attribute 'hide'}
	Out											: Tc2_MC2.ST_McOutputs;
END_VAR
mcGearOut( 			Slave						:= Axis, 
					Execute						:= TRUE, 
					Done						=> Out.Done, 
					Busy						=> Out.Busy, 
					Error						=> Out.Error, 
					ErrorID						=> Out.ErrorID);

					
pGear 											REF= Out;

GearOutEx										:= TRUE;
END_METHOD

METHOD Halt 									: REFERENCE TO Tc2_MC2.ST_McOutputs
VAR_INPUT
	bExecute									: BOOL;
END_VAR
IF bExecute THEN
	HaltEx();
ELSE
	HaltClear();
END_IF

Halt											REF= pHalt;
END_METHOD

METHOD HaltClear 								: BOOL
VAR
	{attribute 'hide'}
	Out											: Tc2_MC2.ST_McOutputs;
END_VAR
mcHalt(				Axis						:= Axis, 
					Execute						:= FALSE, 
					Done						=> Out.Done, 
					Busy						=> Out.Busy, 
					Active						=> Out.Active, 
					CommandAborted				=> Out.CommandAborted, 
					Error						=> Out.Error, 
					ErrorID						=> Out.ErrorID);

pHalt				 							REF= Out;

HaltClear										:= TRUE;
END_METHOD

METHOD HaltEx 									: BOOL
VAR
	{attribute 'hide'}
	Out											: Tc2_MC2.ST_McOutputs;
END_VAR
mcHalt(				Axis						:= Axis, 
					Execute						:= TRUE, 
					Deceleration				:= fDeceleration, 
					Jerk						:= fJerk, 
					BufferMode					:= eBufferMode,
					Options						:= , 
					Done						=> Out.Done, 
					Busy						=> Out.Busy, 
					Active						=> Out.Active, 
					CommandAborted				=> Out.CommandAborted, 
					Error						=> Out.Error, 
					ErrorID						=> Out.ErrorID);

pHalt				 							REF= Out;

HaltEx											:= TRUE;
END_METHOD

METHOD Home 									: REFERENCE TO Tc2_MC2.ST_McOutputs
VAR_INPUT
	bExecute									: BOOL;
	bCalibrationCam								: BOOL;
	eHomingMode									: Tc2_MC2.MC_HomingMode;
END_VAR
IF bExecute THEN
	HomeEx(bCalibrationCam := bCalibrationCam, eHomingMode := eHomingMode);
ELSE
	HomeClear(bCalibrationCam := bCalibrationCam);
END_IF

Home											REF= pHome;
END_METHOD

METHOD HomeClear 								: BOOL
VAR_INPUT
	bCalibrationCam								: BOOL;
END_VAR
VAR
	{attribute 'hide'}
	Out											: Tc2_MC2.ST_McOutputs;
END_VAR
mcHome(				Axis						:= Axis, 
					Execute						:= FALSE, 
					bCalibrationCam				:= bCalibrationCam, 
					Done						=> Out.Done, 
					Busy						=> Out.Busy, 
					Active						=> Out.Active, 
					CommandAborted				=> Out.CommandAborted, 
					Error						=> Out.Error, 
					ErrorID						=> Out.ErrorID);
					
pHome 											REF= Out;
pOut											REF= Out;

HomeClear										:= TRUE;
END_METHOD

METHOD HomeDefault 								: REFERENCE TO Tc2_MC2.ST_McOutputs
VAR_INPUT
	bExecute									: BOOL;
	bCalibrationCam								: BOOL;
END_VAR
Home(bExecute := bExecute, bCalibrationCam := bCalibrationCam, eHomingMode := Tc2_MC2.MC_HomingMode.MC_DefaultHoming);

HomeDefault										REF= pHome;
END_METHOD

METHOD HomeDefaultPos0 							: REFERENCE TO Tc2_MC2.ST_McOutputs
VAR_INPUT
	bExecute									: BOOL;
	bCalibrationCam								: BOOL;
END_VAR
fPosition 										:= 0.0;
Home(bExecute := bExecute, bCalibrationCam := bCalibrationCam, eHomingMode := Tc2_MC2.MC_HomingMode.MC_DefaultHoming);

HomeDefaultPos0									REF= pHome;
END_METHOD

METHOD HomeDirect 								: REFERENCE TO Tc2_MC2.ST_McOutputs
VAR_INPUT
	bExecute									: BOOL;
END_VAR
Home(bExecute := bExecute, bCalibrationCam := FALSE, eHomingMode := Tc2_MC2.MC_HomingMode.MC_Direct);

HomeDirect										REF= pHome;
END_METHOD

METHOD HomeEx 									: BOOL
VAR_INPUT
	bCalibrationCam								: BOOL;
	eHomingMode									: Tc2_MC2.MC_HomingMode;
END_VAR
VAR
	{attribute 'hide'}
	Out											: Tc2_MC2.ST_McOutputs;
END_VAR
mcHome(				Axis						:= Axis, 
					Execute						:= TRUE, 
					Position					:= fPosition,  
					HomingMode					:= eHomingMode, 
					BufferMode					:= , 
					Options						:= , 
					bCalibrationCam				:= bCalibrationCam, 
					Done						=> Out.Done, 
					Busy						=> Out.Busy, 
					Active						=> Out.Active, 
					CommandAborted				=> Out.CommandAborted, 
					Error						=> Out.Error, 
					ErrorID						=> Out.ErrorID);
					
pHome 											REF= Out;
pOut											REF= Out;

HomeEx											:= TRUE;
END_METHOD

METHOD HomeForceCalibration 					: REFERENCE TO Tc2_MC2.ST_McOutputs
VAR_INPUT
	bExecute									: BOOL;
END_VAR
Home(bExecute := bExecute, bCalibrationCam := FALSE, eHomingMode := Tc2_MC2.MC_HomingMode.MC_ForceCalibration);

HomeForceCalibration							REF= pHome;
END_METHOD

METHOD HomeResetCalibration 					: REFERENCE TO Tc2_MC2.ST_McOutputs
VAR_INPUT
	bExecute									: BOOL;
END_VAR
Home(bExecute := bExecute, bCalibrationCam := FALSE, eHomingMode := Tc2_MC2.MC_HomingMode.MC_ResetCalibration);

HomeResetCalibration							REF= pHome;
END_METHOD

METHOD PROTECTED Init 							: BOOL
VAR_INST
	{attribute 'hide'}
	nStep										: DINT;
	{attribute 'hide'}
	fbGetCurTaskIdx								: Tc2_System.GETCURTASKINDEX;
	{attribute 'hide'}
	nOnlineChangeCntOld							: UDINT;
END_VAR
VAR
	{attribute 'hide'}
	Out											: Tc2_MC2.ST_McOutputs;
	{attribute 'hide'}
	bOnlineChangeDetected						: BOOL;
END_VAR
CASE nStep OF
	
	0:	// Init
	
		fbGetCurTaskIdx();
		IF _TaskInfo[fbGetCurTaskIdx.index].FirstCycle THEN
			nStep								:= nStep + 10;
		END_IF

	10: // Nc Axis is alive?
	
		IF Axis.NcToPlc.StateDWord <> 0 THEN
			nStep								:= nStep + 10;
		END_IF
		
	20: // 

		Out := ReadParameterSet(bExecute := TRUE);
		nStep									:= nStep + 10;
		
	30: //

		Out := ReadParameterSet(bExecute := TRUE);
		IF Out.Done THEN
			Out := ReadParameterSet(bExecute := FALSE);
			nStep								:= 100;
		ELSIF Out.Error THEN
			Out := ReadParameterSet(bExecute := FALSE);
			nStep								:= nStep - 10;
		END_IF

	100:
	
		Init									:= TRUE;
		
		// Online change detection
		bOnlineChangeDetected					:= nOnlineChangeCntOld <> _AppInfo.OnlineChangeCnt;
		IF bOnlineChangeDetected THEN
			nStep 								:= 20;
		END_IF
		nOnlineChangeCntOld 					:= _AppInfo.OnlineChangeCnt;

END_CASE
END_METHOD

METHOD IsConsequentialError 					: BOOL
VAR CONSTANT
	// Filtered Errors
	nConsequentialError							: UDINT 	:= 16#42A0; (*Group/axis consequential error" Consequential error resulting from another causative error 
																		related to another axis within the group. 
																		Group/axis consequential errors can occur in relation to master/slave couplings or 
																		with multiple axis interpolating DXD groups. 
																		If, for instance, it is detected that the following error limit of a master axis has been exceeded, 
																		then this consequential error is assigned to all the other master axes and slave axes in this group.*)
END_VAR
VAR_INPUT
	nErrorID									: UDINT;
END_VAR
IsConsequentialError 							:= nErrorID = nConsequentialError;
END_METHOD

METHOD Jog 										: REFERENCE TO Tc2_MC2.ST_McOutputs
VAR_INPUT
	bFw											: BOOL;
	bBw											: BOOL;
END_VAR
VAR_INST
	{attribute 'hide'}
	nStep										: DINT;
END_VAR
CASE nStep OF
	
	0:	
	
		IF bFw THEN
			JogFwEx();
			IF NOT pJog.Error THEN
				nStep							:= 100;
			END_IF
		ELSIF bBw THEN
			JogBwEx();
			IF NOT pJog.Error THEN
				nStep							:= 200;
			END_IF
		ELSE
			JogClear();
		END_IF
	
	100: // Fwd execution, stop or change

		IF bFw THEN
			JogFwEx();
			IF NOT pJog.Busy THEN
				nStep							:= nStep + 10;
			END_IF
		ELSE
			JogClear();
			nStep								:= 300;
		END_IF
			
	110: // Move finished - wait till move command removed

		IF bFw THEN
			JogFwEx();
		ELSE
			IF bBw THEN
				JogBwEx();
				IF NOT pJog.Error THEN
					nStep						:= 200;
				ELSE
					nStep						:= 0;
				END_IF
			ELSE
				JogClear();
				nStep							:= 0;			
			END_IF
		END_IF
	
	200: // Bwd execution, stop or change

		IF bBw THEN
			JogBwEx();
			IF NOT pJog.Busy THEN
				nStep							:= nStep + 10;
			END_IF
		ELSE
			JogClear();
			nStep								:= 300;
		END_IF
 			
	210: // Move finished - wait till move command removed

		IF bBw THEN
			JogBwEx();
		ELSE
			IF bFw THEN
				JogFwEx();
				IF NOT pJog.Error THEN
					nStep						:= 100;
				ELSE
					nStep						:= 0;
				END_IF
			ELSE
				JogClear();
				nStep							:= 0;			
			END_IF
		END_IF
 			
	300: // Moving, no command - wait till move end
	
		JogClear();
		IF NOT pJog.Busy THEN
			nStep							:= 0;		
		END_IF
		
END_CASE

Jog												REF= pJog;
END_METHOD

METHOD JogBwEx 									: BOOL
VAR
	{attribute 'hide'}
	Out											: Tc2_MC2.ST_McOutputs;
END_VAR
mcJog(				Axis						:= Axis, 
					JogForward					:= FALSE, 
					JogBackwards				:= TRUE, 
					Mode						:= eJogMode, 
					Position					:= fPosition, 
					Velocity					:= fVelocity, 
					Acceleration				:= fAcceleration, 
					Deceleration				:= fDeceleration, 
					Jerk						:= fJerk,
					Done						=> Out.Done, 
					Busy						=> Out.Busy, 
					Active						=> Out.Active, 
					CommandAborted				=> Out.CommandAborted, 
					Error						=> Out.Error, 
					ErrorID						=> Out.ErrorID);

	
pJog	 										REF= Out;
pOut											REF= Out;

JogBwEx											:= TRUE;
END_METHOD

METHOD JogClear 								: BOOL
VAR
	{attribute 'hide'}
	Out											: Tc2_MC2.ST_McOutputs;
END_VAR
mcJog(				Axis						:= Axis, 
					JogForward					:= FALSE, 
					JogBackwards				:= FALSE, 
					Done						=> Out.Done, 
					Busy						=> Out.Busy, 
					Active						=> Out.Active, 
					CommandAborted				=> Out.CommandAborted, 
					Error						=> Out.Error, 
					ErrorID						=> Out.ErrorID);

	
pJog	 										REF= Out;
pOut											REF= Out;

JogClear										:= TRUE;
END_METHOD

METHOD JogContinous 							: REFERENCE TO Tc2_MC2.ST_McOutputs
VAR_INPUT
	bFw											: BOOL;
	bBw											: BOOL;
END_VAR
eJogMode										:= Tc2_MC2.E_JogMode.MC_JOGMODE_CONTINOUS;

Jog(bFw := bFw, bBw	:= bBw);

JogContinous									REF= pJog;
END_METHOD

METHOD JogFast 									: REFERENCE TO Tc2_MC2.ST_McOutputs
VAR_INPUT
	bFw											: BOOL;
	bBw											: BOOL;
END_VAR
eJogMode										:= Tc2_MC2.E_JogMode.MC_JOGMODE_STANDARD_FAST;

Jog(bFw := bFw, bBw	:= bBw);

JogFast											REF= pJog;
END_METHOD

METHOD JogFwEx 									: BOOL
VAR
	{attribute 'hide'}
	Out											: Tc2_MC2.ST_McOutputs;
END_VAR
mcJog(				Axis						:= Axis, 
					JogForward					:= TRUE, 
					JogBackwards				:= FALSE, 
					Mode						:= eJogMode, 
					Position					:= fPosition, 
					Velocity					:= fVelocity, 
					Acceleration				:= fAcceleration, 
					Deceleration				:= fDeceleration, 
					Jerk						:= fJerk,
					Done						=> Out.Done, 
					Busy						=> Out.Busy, 
					Active						=> Out.Active, 
					CommandAborted				=> Out.CommandAborted, 
					Error						=> Out.Error, 
					ErrorID						=> Out.ErrorID);

	
pJog	 										REF= Out;
pOut											REF= Out;

JogFwEx											:= TRUE;
END_METHOD

METHOD JogInching 								: REFERENCE TO Tc2_MC2.ST_McOutputs
VAR_INPUT
	bFw											: BOOL;
	bBw											: BOOL;
END_VAR
eJogMode										:= Tc2_MC2.E_JogMode.MC_JOGMODE_INCHING;

Jog(bFw := bFw, bBw	:= bBw);

JogInching										REF= pJog;
END_METHOD

METHOD JogInchingModulo 						: REFERENCE TO Tc2_MC2.ST_McOutputs
VAR_INPUT
	bFw											: BOOL;
	bBw											: BOOL;
END_VAR
eJogMode										:= Tc2_MC2.E_JogMode.MC_JOGMODE_INCHING_MODULO;

Jog(bFw := bFw, bBw	:= bBw);

JogInchingModulo								REF= pJog;
END_METHOD

METHOD JogSlow 									: REFERENCE TO Tc2_MC2.ST_McOutputs
VAR_INPUT
	bFw											: BOOL;
	bBw											: BOOL;
END_VAR
eJogMode										:= Tc2_MC2.E_JogMode.MC_JOGMODE_STANDARD_SLOW;

Jog(bFw := bFw, bBw	:= bBw);

JogSlow											REF= pJog;
END_METHOD

METHOD LagMonitoringDisable 					: REFERENCE TO Tc2_MC2.ST_McOutputs
VAR_INPUT
	bExecute									: BOOL;
END_VAR
VAR
	{attribute 'hide'}
	Out											: Tc2_MC2.ST_McOutputs;
END_VAR
fbPosLagMonitoring.bState						:= FALSE;

Out := fbPosLagMonitoring.WriteState(bExecute 	:= bExecute, 
									nAxisID 	:= Axis.NcToPlc.AxisId);

//pWriteLimitSwitch								REF= Out;

LagMonitoringDisable							REF= Out;
END_METHOD

METHOD LagMonitoringEnable 						: REFERENCE TO Tc2_MC2.ST_McOutputs
VAR_INPUT
	bExecute									: BOOL;
END_VAR
VAR
	{attribute 'hide'}
	Out											: Tc2_MC2.ST_McOutputs;
END_VAR
fbPosLagMonitoring.bState						:= TRUE;

Out := fbPosLagMonitoring.WriteState(bExecute 	:= bExecute, 
									nAxisID 	:= Axis.NcToPlc.AxisId);

//pWriteLimitSwitch								REF= Out;

LagMonitoringEnable								REF= Out;
END_METHOD

METHOD LimitSwitchDisable 						: REFERENCE TO Tc2_MC2.ST_McOutputs
VAR_INPUT
	bExecute									: BOOL;
END_VAR
VAR
	{attribute 'hide'}
	Out											: Tc2_MC2.ST_McOutputs;
END_VAR
VAR_INST
	{attribute 'hide'}
	nStep										: DINT;
END_VAR
CASE nStep OF

	0: 
		IF bExecute THEN
			nStep								:= nStep + 5;
		END_IF
		
	5:

		Out := LimitSwitchDisableMax(bExecute := TRUE);
		IF Out.Busy THEN
			nStep								:= nStep + 5;
		END_IF
	
	10:
	
		Out := LimitSwitchDisableMax(bExecute := FALSE);
		IF Out.Done THEN
			nStep								:= nStep + 5;
		ELSIF Out.Error THEN
			nStep								:= nStep + 10_000;
		END_IF
	
	15: 
	
		Out := LimitSwitchDisableMin(bExecute := TRUE);
		IF Out.Busy THEN
			nStep								:= nStep + 5;
		END_IF
		
	20:
	
		Out := LimitSwitchDisableMin(bExecute := FALSE);
		IF Out.Done THEN
			nStep								:= 100;
		ELSIF Out.Error THEN
			nStep								:= nStep + 10_000;
		END_IF
		
	100:
	
		Out.Done								:= TRUE;
		IF bExecute THEN
			nStep								:= nStep + 1;
		ELSE
			nStep								:= 0;
		END_IF
		
	101:
	
		Out.Done								:= TRUE;	
		IF NOT bExecute THEN
			Out.Done							:= FALSE;
			nStep								:= 0;
		END_IF
			
	10_000..10_099:
	
		Out.Error								:= TRUE;
		IF bExecute THEN
			nStep								:= nStep + 100;
		ELSE
			nStep								:= 0;
		END_IF
		
	10_100..10_199:
	
		Out.Error								:= TRUE;	
		IF NOT bExecute THEN
			Out.Error							:= FALSE;
			nStep								:= 0;
		END_IF	

END_CASE

Out.Busy 										:= nStep <> 0 
													AND NOT Out.Done 
													AND NOT Out.Error;
													
LimitSwitchDisable								REF= Out;
END_METHOD

METHOD LimitSwitchDisableMax 					: REFERENCE TO Tc2_MC2.ST_McOutputs
VAR_INPUT
	bExecute									: BOOL;
END_VAR
VAR
	{attribute 'hide'}
	Out											: Tc2_MC2.ST_McOutputs;
END_VAR
fbLimitSwitch.LimitSwitchStateMax				:= FALSE;

Out := fbLimitSwitch.WriteStateMax(	bExecute 	:= bExecute, 
									nAxisID 	:= Axis.NcToPlc.AxisId);

pLimitSwitch									REF= Out;

LimitSwitchDisableMax							REF= Out;
END_METHOD

METHOD LimitSwitchDisableMin 					: REFERENCE TO Tc2_MC2.ST_McOutputs
VAR_INPUT
	bExecute									: BOOL;
END_VAR
VAR
	{attribute 'hide'}
	Out											: Tc2_MC2.ST_McOutputs;
END_VAR
fbLimitSwitch.LimitSwitchStateMin				:= FALSE;

Out := fbLimitSwitch.WriteStateMin(	bExecute 	:= bExecute, 
									nAxisID 	:= Axis.NcToPlc.AxisId);

pLimitSwitch									REF= Out;

LimitSwitchDisableMin							REF= Out;
END_METHOD

METHOD LimitSwitchEnable 						: REFERENCE TO Tc2_MC2.ST_McOutputs
VAR_INPUT
	bExecute									: BOOL;
END_VAR
VAR
	{attribute 'hide'}
	Out											: Tc2_MC2.ST_McOutputs;
END_VAR
VAR_INST
	{attribute 'hide'}
	nStep										: DINT;
END_VAR
CASE nStep OF

	0: 
		IF bExecute THEN
			nStep								:= nStep + 5;
		END_IF
		
	5:

		Out := LimitSwitchEnableMax(bExecute := TRUE);
		IF Out.Busy THEN
			nStep								:= nStep + 5;
		END_IF
	
	10:
	
		Out := LimitSwitchEnableMax(bExecute := FALSE);
		IF NOT Out.Busy AND NOT Out.Error THEN
			nStep								:= nStep + 1;
		ELSIF Out.Error THEN
			nStep								:= nStep + 10_000;
		END_IF
		
	11:

		LimitSwitchEnableMax(bExecute := FALSE);
		nStep									:= nStep + 4;
	
	15: 
	
		Out := LimitSwitchEnableMin(bExecute := TRUE);
		IF Out.Busy THEN
			nStep								:= nStep + 5;
		END_IF
		
	20:
	
		Out := LimitSwitchEnableMin(bExecute := FALSE);
		IF NOT Out.Busy AND NOT Out.Error THEN
			nStep								:= nStep + 1;
		ELSIF Out.Error THEN
			nStep								:= nStep + 10_000;
		END_IF
			
	21:

		LimitSwitchEnableMin(bExecute := FALSE);
		nStep									:= 100;
		
	100:
	
		Out.Done								:= TRUE;
		IF bExecute THEN
			nStep								:= nStep + 1;
		ELSE
			nStep								:= 0;
		END_IF
		
	101:
	
		Out.Done								:= TRUE;	
		IF NOT bExecute THEN
			Out.Done							:= FALSE;
			nStep								:= 0;
		END_IF
			
	10_000..10_099:
	
		Out.Error								:= TRUE;
		IF bExecute THEN
			nStep								:= nStep + 100;
		ELSE
			nStep								:= 0;
		END_IF
		
	10_100..10_199:
	
		Out.Error								:= TRUE;	
		IF NOT bExecute THEN
			Out.Error							:= FALSE;
			nStep								:= 0;
		END_IF	

END_CASE

Out.Busy 										:= nStep <> 0 
													AND NOT Out.Done 
													AND NOT Out.Error;
													
LimitSwitchEnable								REF= Out;
END_METHOD

METHOD LimitSwitchEnableMax 					: REFERENCE TO Tc2_MC2.ST_McOutputs
VAR_INPUT
	bExecute									: BOOL;
END_VAR
VAR
	{attribute 'hide'}
	Out											: Tc2_MC2.ST_McOutputs;
END_VAR
fbLimitSwitch.LimitSwitchStateMax				:= TRUE;

Out := fbLimitSwitch.WriteStateMax(	bExecute 	:= bExecute, 
									nAxisID 	:= Axis.NcToPlc.AxisId);

pLimitSwitch									REF= Out;

LimitSwitchEnableMax							REF= Out;
END_METHOD

METHOD LimitSwitchEnableMin 					: REFERENCE TO Tc2_MC2.ST_McOutputs
VAR_INPUT
	bExecute									: BOOL;
END_VAR
VAR
	{attribute 'hide'}
	Out											: Tc2_MC2.ST_McOutputs;
END_VAR
fbLimitSwitch.LimitSwitchStateMin				:= TRUE;

Out := fbLimitSwitch.WriteStateMin(	bExecute 	:= bExecute, 
									nAxisID 	:= Axis.NcToPlc.AxisId);

pLimitSwitch									REF= Out;

LimitSwitchEnableMin							REF= Out;
END_METHOD

METHOD LimitSwitchRead 							: REFERENCE TO Tc2_MC2.ST_McOutputs
VAR_INPUT
	bExecute									: BOOL;
END_VAR
LimitSwitchRead := fbLimitSwitch.ReadParams(	bExecute 	:= bExecute, 
												nAxisID 	:= Axis.NcToPlc.AxisId);
												
fLimitSwitchPositionMin							:= fbLimitSwitch.LimitSwitchPositionMin;
fLimitSwitchPositionMax							:= fbLimitSwitch.LimitSwitchPositionMax;
bLimitSwitchStateMin							:= fbLimitSwitch.LimitSwitchStateMin;
bLimitSwitchStateMax							:= fbLimitSwitch.LimitSwitchStateMax;
END_METHOD

METHOD LimitSwitchReadStateMax 					: REFERENCE TO Tc2_MC2.ST_McOutputs
VAR_INPUT
	bExecute									: BOOL;
END_VAR
pLimitSwitch := fbLimitSwitch.ReadStateMax(
									bExecute 	:= bExecute, 
									nAxisID 	:= Axis.NcToPlc.AxisId);

LimitSwitchReadStateMax							REF= pLimitSwitch;

bLimitSwitchStateMax							:= fbLimitSwitch.LimitSwitchStateMax;
END_METHOD

METHOD LimitSwitchReadStateMin 					: REFERENCE TO Tc2_MC2.ST_McOutputs
VAR_INPUT
	bExecute									: BOOL;
END_VAR
pLimitSwitch := fbLimitSwitch.ReadStateMin(
									bExecute 	:= bExecute, 
									nAxisID 	:= Axis.NcToPlc.AxisId);

LimitSwitchReadStateMin							REF= pLimitSwitch;

bLimitSwitchStateMin							:= fbLimitSwitch.LimitSwitchStateMin;
END_METHOD

METHOD LimitSwitchReadValueMax 					: REFERENCE TO Tc2_MC2.ST_McOutputs
VAR_INPUT
	bExecute									: BOOL;
END_VAR
pLimitSwitch := fbLimitSwitch.ReadValueMax(
									bExecute 	:= bExecute, 
									nAxisID 	:= Axis.NcToPlc.AxisId);

LimitSwitchReadValueMax							REF= pLimitSwitch;

fLimitSwitchPositionMax							:= fbLimitSwitch.LimitSwitchPositionMax;
END_METHOD

METHOD LimitSwitchReadValueMin 					: REFERENCE TO Tc2_MC2.ST_McOutputs
VAR_INPUT
	bExecute									: BOOL;
END_VAR
pLimitSwitch := fbLimitSwitch.ReadValueMin(
									bExecute 	:= bExecute, 
									nAxisID 	:= Axis.NcToPlc.AxisId);

LimitSwitchReadValueMin							REF= pLimitSwitch;

fLimitSwitchPositionMin							:= fbLimitSwitch.LimitSwitchPositionMin;
END_METHOD

METHOD LimitSwitchWrite 						: REFERENCE TO Tc2_MC2.ST_McOutputs
VAR_INPUT
	bExecute									: BOOL;
END_VAR
VAR
	{attribute 'hide'}
	Out											: Tc2_MC2.ST_McOutputs;
END_VAR
fbLimitSwitch.LimitSwitchPositionMin			:= fLimitSwitchPositionMin;
fbLimitSwitch.LimitSwitchPositionMax			:= fLimitSwitchPositionMax;
fbLimitSwitch.LimitSwitchStateMin				:= bLimitSwitchStateMin;
fbLimitSwitch.LimitSwitchStateMax				:= bLimitSwitchStateMax;

Out := fbLimitSwitch.WriteParams(	bExecute 	:= bExecute, 
												nAxisID 	:= Axis.NcToPlc.AxisId);
												
LimitSwitchWrite 								REF= Out;
END_METHOD

METHOD LimitSwitchWriteMax 						: REFERENCE TO Tc2_MC2.ST_McOutputs
VAR_INPUT
	bExecute									: BOOL;
END_VAR
VAR
	{attribute 'hide'}
	Out											: Tc2_MC2.ST_McOutputs;
END_VAR
fbLimitSwitch.LimitSwitchPositionMax			:= fLimitSwitchPositionMax;

Out := fbLimitSwitch.WriteValueMax(	bExecute 	:= bExecute, 
									nAxisID 	:= Axis.NcToPlc.AxisId);

pLimitSwitch									REF= Out;

LimitSwitchWriteMax								REF= Out;
END_METHOD

METHOD LimitSwitchWriteMin 						: REFERENCE TO Tc2_MC2.ST_McOutputs
VAR_INPUT
	bExecute									: BOOL;
END_VAR
VAR
	{attribute 'hide'}
	Out											: Tc2_MC2.ST_McOutputs;
END_VAR
fbLimitSwitch.LimitSwitchPositionMin			:= fLimitSwitchPositionMin;

Out := fbLimitSwitch.WriteValueMin(	bExecute 	:= bExecute, 
									nAxisID 	:= Axis.NcToPlc.AxisId);

pLimitSwitch									REF= Out;

LimitSwitchWriteMin								REF= Out;
END_METHOD

METHOD Manual			 						: BOOL
VAR_INPUT
	stManual									: REFERENCE TO ST_AxisControlManual;
END_VAR
VAR_INST
	{attribute 'hide'}
	bManualRefError								: BOOL;
END_VAR
IF NOT __ISVALIDREF(stManual) THEN

	IF NOT bManualRefError THEN
		ADSLOGSTR(ADSLOG_MSGTYPE_ERROR,'FB_AxisBase critical error - Manual Reference not assigned! FB instance: %s',sInstancePath);
	END_IF

	bManualRefError								:= TRUE;
	
	RETURN;

END_IF

bManualRefError									:= FALSE;
fVelocity										:= stManual.fVelocity;
fPosition										:= stManual.fPosition;
fOverride										:= stManual.fOverride;
bEnable											:= stManual.bEnable;
Stop(bExecute									:= stManual.bStop);
Reset(bExecute									:= stManual.bReset);

// Absolute/modulo
IF stManual.bModulo THEN
	MoveAbsoluteClear();
	MoveModuloShort(bExecute := stManual.bExecute);
ELSE
	MoveModuloClear();
	MoveAbsolute(bExecute := stManual.bExecute);
END_IF

// Jog mode
IF stManual.bSlowForward OR stManual.bSlowBackward THEN
	JogSlow(bFw := stManual.bSlowForward, bBw := stManual.bSlowBackward);
ELSIF stManual.bFastForward OR stManual.bFastBackward THEN
	JogFast(bFw := stManual.bFastForward, bBw := stManual.bFastBackward);
ELSE
	JogClear();
END_IF

Manual											:= TRUE;
END_METHOD

METHOD Manual_1 									: BOOL
VAR_INST
	nStep										: DINT;
END_VAR
VAR
	Out											: Tc2_MC2.ST_McOutputs;
END_VAR
ManualRead(stManual);

CASE nStep OF
	
	0:
	
		IF stManual.bEnableManualMode THEN
			stManual.lrOverride 				:= fOverride;
			Out									:= pPower;
			stManual.bEnable					:= Out.Busy;
			Manual(stManual := stManual);
			nStep								:= nStep + 10;
		END_IF
		
	10: 
	
		Manual(stManual := stManual);
		IF NOT stManual.bEnableManualMode THEN
			ClearAll();
			stManual.bExecute					:= FALSE;
			stManual.bLockBrake					:= FALSE;
			stManual.bReleaseBrake				:= FALSE;
			IF stManual.stStatus.Moving THEN
				Stop(bExecute := TRUE);
				nStep							:= nStep + 10;
			ELSE
				nStep							:= 100;
			END_IF
		END_IF
		
	20:
	
		Out := Stop(bExecute := FALSE);
		IF NOT Out.Busy THEN
			nStep								:= 100;
		END_IF
		
	100:
	
		nStep									:= 0;	
		
END_CASE


Manual 											:= nStep <> 0;
END_METHOD

METHOD PRIVATE ManualEx_1 						: BOOL
VAR
	OutReadLS									: Tc2_MC2.ST_McOutputs;
	OutWriteLS									: Tc2_MC2.ST_McOutputs;
END_VAR
//CheckAxisRef();
(*
Velocity										:= stManual.lrVelocity;
Position										:= stManual.lrPosition;
IF stManual.lrOverride > 0.1 THEN
	Override									:= stManual.lrOverride;
ELSE
	stManual.lrOverride							:= Override;
END_IF
Power(bEnable									:= stManual.bEnable);
Halt(bExecute									:= stManual.bStop);
Reset(bExecute									:= stManual.bReset);

// Absolute/modulo
IF stManual.bModulo THEN
	MoveAbsoluteClear();
	MoveModuloShort(bExecute := stManual.bExecute);	
	stManual.lrActPosVisu 						:= Axis.NcToPlc.ModuloActPos;
	stManual.lrSetPosVisu 						:= Axis.NcToPlc.ModuloSetPos;
ELSE
	MoveModuloClear();
	MoveAbsolute(bExecute := stManual.bExecute);
	stManual.lrActPosVisu 						:= Axis.NcToPlc.ActPos;
	stManual.lrSetPosVisu 						:= Axis.NcToPlc.SetPos;	
END_IF

// Jog mode
IF stManual.bSlowForward OR stManual.bSlowBackward THEN
	JogSlow(bFw := stManual.bSlowForward, bBw := stManual.bSlowBackward);
ELSIF stManual.bFastForward OR stManual.bFastBackward THEN
	JogFast(bFw := stManual.bFastForward, bBw := stManual.bFastBackward);
ELSE
	JogClear();
END_IF

// Limit switches
OutReadLS 		:= LimitSwitchRead(bExecute := stManual.bReadLS);
IF OutReadLS.Done THEN
	stManual.lrLimitSwitchPositionMax 			:= LimitSwitchPositionMax;
	stManual.lrLimitSwitchPositionMin 			:= LimitSwitchPositionMin;
	stManual.bLimitSwitchStateMax 				:= LimitSwitchStateMax;
	stManual.bLimitSwitchStateMin 				:= LimitSwitchStateMin;
END_IF
IF stManual.bWriteLS THEN
	LimitSwitchPositionMax 						:= stManual.lrLimitSwitchPositionMax;
	LimitSwitchPositionMin 						:= stManual.lrLimitSwitchPositionMin;
	LimitSwitchStateMax 						:= stManual.bLimitSwitchStateMax;
	LimitSwitchStateMin 						:= stManual.bLimitSwitchStateMin;
END_IF
OutWriteLS 		:= LimitSwitchWrite(bExecute := stManual.bWriteLS);


// States

stManual.stStatus								:= Axis.Status;

stManual.bError									:= Axis.Status.Error;
stManual.nErrorID								:= Axis.Status.ErrorID;

stManual.lrActPos								:= Axis.NcToPlc.ActPos;
stManual.lrModuloActPos							:= Axis.NcToPlc.ModuloActPos;
stManual.lrActVelo								:= Axis.NcToPlc.ActVelo;
stManual.lrActTorque							:= Axis.NcToPlc.ActTorque;
stManual.lrSetPos								:= Axis.NcToPlc.SetPos;
stManual.lrModuloSetPos							:= Axis.NcToPlc.ModuloSetPos;
stManual.lrSetVelo								:= Axis.NcToPlc.SetVelo;
stManual.lrPosDiff								:= Axis.NcToPlc.PosDiff;
stManual.bConsequentialError					:= ConsequentialError;

ManualEx_1										:= TRUE;

*)
END_METHOD

METHOD PRIVATE ManualEx_2 						: BOOL
VAR_INPUT
	stManual									: REFERENCE TO ST_AxisControlManualBase;
END_VAR
VAR
	OutReadLS									: Tc2_MC2.ST_McOutputs;
	OutWriteLS									: Tc2_MC2.ST_McOutputs;
END_VAR
VAR_INST
	bManualRefError								: BOOL;
END_VAR
IF NOT __ISVALIDREF(stManual) THEN

	IF NOT bManualRefError THEN
		ADSLOGSTR(ADSLOG_MSGTYPE_ERROR,'FB_AxisBase critical error - Manual Reference not assigned! FB instance: %s',sInstancePath);
	END_IF

	bManualRefError								:= TRUE;
	
	RETURN;

END_IF

bManualRefError									:= FALSE;
fVelocity										:= stManual.lrVelocity;
fPosition										:= stManual.lrPosition;
fOverride										:= stManual.lrOverride;
Power(bEnable									:= stManual.bEnable);
Halt(bExecute									:= stManual.bStop);
Reset(bExecute									:= stManual.bReset);

// Absolute/modulo
IF stManual.bModulo THEN
	MoveAbsoluteClear();
	MoveModuloShort(bExecute := stManual.bExecute);
ELSE
	MoveModuloClear();
	MoveAbsolute(bExecute := stManual.bExecute);
END_IF

// Jog mode
IF stManual.bSlowForward OR stManual.bSlowBackward THEN
	JogSlow(bFw := stManual.bSlowForward, bBw := stManual.bSlowBackward);
ELSIF stManual.bFastForward OR stManual.bFastBackward THEN
	JogFast(bFw := stManual.bFastForward, bBw := stManual.bFastBackward);
ELSE
	JogClear();
END_IF

// Limit switches
OutReadLS 		:= LimitSwitchRead(bExecute := stManual.bReadLS);
IF OutReadLS.Done THEN
	stManual.lrLimitSwitchPositionMax 			:= fLimitSwitchPositionMax;
	stManual.lrLimitSwitchPositionMin 			:= fLimitSwitchPositionMin;
	stManual.bLimitSwitchStateMax 				:= bLimitSwitchStateMax;
	stManual.bLimitSwitchStateMin 				:= bLimitSwitchStateMin;
END_IF
IF stManual.bWriteLS THEN
	fLimitSwitchPositionMax 						:= stManual.lrLimitSwitchPositionMax;
	fLimitSwitchPositionMin 						:= stManual.lrLimitSwitchPositionMin;
	bLimitSwitchStateMax 						:= stManual.bLimitSwitchStateMax;
	bLimitSwitchStateMin 						:= stManual.bLimitSwitchStateMin;
END_IF
OutWriteLS 		:= LimitSwitchWrite(bExecute := stManual.bWriteLS);

Manual										:= TRUE;
END_METHOD

METHOD ManualHMI 								: BOOL
VAR_INPUT
	bEnable										: BOOL;
END_VAR
VAR_INST
	{attribute 'hide'}
	nStep										: DINT;
END_VAR
VAR
	{attribute 'hide'}
	PowerOut									: Tc2_MC2.ST_McOutputs;
END_VAR
ManualRead(); 									// Read data neccesary for HMI

// Absolute/modulo display
IF stManualHMI.stCommands.bModulo THEN
	stManualHMI.fActPos 						:= Axis.NcToPlc.ModuloActPos;
	stManualHMI.fSetPos 						:= Axis.NcToPlc.ModuloSetPos;
ELSE
	stManualHMI.fActPos 						:= Axis.NcToPlc.ActPos;
	stManualHMI.fSetPos 						:= Axis.NcToPlc.SetPos;	
END_IF

CASE nStep OF
	
	0:
	
		IF bEnable THEN
			// Gentle mode switch
			PowerOut							:= pPower;
			stManualHMI.stCommands.bEnable		:= PowerOut.Busy;
			stManualHMI.stCommands.fOverride	:= fOverride;
			Manual(stManual := stManualHMI.stCommands);

			nStep								:= nStep + 10;
		END_IF
	
	10:
	
		Manual(stManual := stManualHMI.stCommands);
	
		IF NOT bEnable AND bNotMoving THEN
			nStep								:= 0;
		END_IF	

END_CASE

ManualHMI										:= nStep <> 0;
END_METHOD

METHOD PRIVATE ManualRead 						: BOOL
stManualHMI.bError								:= Axis.Status.Error;
stManualHMI.nErrorID							:= Axis.Status.ErrorID;

stManualHMI.fActPos								:= Axis.NcToPlc.ActPos;
stManualHMI.fModuloActPos						:= Axis.NcToPlc.ModuloActPos;
stManualHMI.fActVelo							:= Axis.NcToPlc.ActVelo;
stManualHMI.fActTorque							:= Axis.NcToPlc.ActTorque;
stManualHMI.fSetPos								:= Axis.NcToPlc.SetPos;
stManualHMI.fModuloSetPos						:= Axis.NcToPlc.ModuloSetPos;
stManualHMI.fSetVelo							:= Axis.NcToPlc.SetVelo;
stManualHMI.fPosDiff							:= Axis.NcToPlc.PosDiff;
stManualHMI.bConsequentialError					:= bConsequentialError;

ManualRead										:= TRUE;
END_METHOD

METHOD PRIVATE ManualVisu 						: BOOL
VAR
	PowerOut									: Tc2_MC2.ST_McOutputs;
END_VAR
// Absolute/modulo
IF stManualVisu.stManual.bModulo THEN
	stManualVisu.lrActPos 						:= Axis.NcToPlc.ModuloActPos;
	stManualVisu.lrSetPos 						:= Axis.NcToPlc.ModuloSetPos;
ELSE
	stManualVisu.lrActPos 						:= Axis.NcToPlc.ActPos;
	stManualVisu.lrSetPos 						:= Axis.NcToPlc.SetPos;	
END_IF

PowerOut										:= pPower;
stManualVisu.bEnable							:= PowerOut.Busy;
stManualVisu.lrOverride							:= fOverride;

ManualVisu										:= TRUE;
END_METHOD

METHOD MoveAbsolute 							: REFERENCE TO Tc2_MC2.ST_McOutputs
VAR_INPUT
	bExecute									: BOOL;
END_VAR
IF bExecute THEN
	MoveAbsoluteEx();
ELSE
	MoveAbsoluteClear();
END_IF

MoveAbsolute									REF= pAbsolute;
END_METHOD

METHOD MoveAbsolute2 							: REFERENCE TO Tc2_MC2.ST_McOutputs
VAR_INPUT
	bExecute									: BOOL;
END_VAR
IF bExecute THEN
	MoveAbsoluteEx2();
ELSE
	MoveAbsoluteClear2();
END_IF

MoveAbsolute2									REF= pAbsolute2;
END_METHOD

METHOD MoveAbsoluteClear 						: BOOL
VAR
	{attribute 'hide'}
	Out											: Tc2_MC2.ST_McOutputs;
END_VAR
mcMoveAbsolute(		Axis						:= Axis, 
					Execute						:= FALSE, 
					Done						=> Out.Done, 
					Busy						=> Out.Busy, 
					Active						=> Out.Active, 
					CommandAborted				=> Out.CommandAborted, 
					Error						=> Out.Error, 
					ErrorID						=> Out.ErrorID);
	
pAbsolute 										REF= Out;
pOut											REF= Out;

MoveAbsoluteClear								:= TRUE;
END_METHOD

METHOD MoveAbsoluteClear2 						: BOOL
VAR
	{attribute 'hide'}
	Out											: Tc2_MC2.ST_McOutputs;
END_VAR
mcMoveAbsolute2(	Axis						:= Axis, 
					Execute						:= FALSE, 
					Done						=> Out.Done, 
					Busy						=> Out.Busy, 
					Active						=> Out.Active, 
					CommandAborted				=> Out.CommandAborted, 
					Error						=> Out.Error, 
					ErrorID						=> Out.ErrorID);
	
pAbsolute2 										REF= Out;
pOut											REF= Out;

MoveAbsoluteClear2								:= TRUE;
END_METHOD

METHOD MoveAbsoluteEx 							: BOOL
VAR
	{attribute 'hide'}
	Out											: Tc2_MC2.ST_McOutputs;
END_VAR
mcMoveAbsolute(		Axis						:= Axis, 
					Execute						:= TRUE, 
					Position					:= fPosition, 
					Velocity					:= fVelocity, 
					Acceleration				:= fAcceleration, 
					Deceleration				:= fDeceleration, 
					Jerk						:= fJerk, 
					BufferMode					:= eBufferMode, 
					Options						:= , 
					Done						=> Out.Done, 
					Busy						=> Out.Busy, 
					Active						=> Out.Active, 
					CommandAborted				=> Out.CommandAborted, 
					Error						=> Out.Error, 
					ErrorID						=> Out.ErrorID);
	
pAbsolute 										REF= Out;
pOut											REF= Out;

MoveAbsoluteEx									:= TRUE;
END_METHOD

METHOD MoveAbsoluteEx2 							: BOOL
VAR
	{attribute 'hide'}
	Out											: Tc2_MC2.ST_McOutputs;
END_VAR
mcMoveAbsolute2(	Axis						:= Axis, 
					Execute						:= TRUE, 
					Position					:= fPosition, 
					Velocity					:= fVelocity, 
					Acceleration				:= fAcceleration, 
					Deceleration				:= fDeceleration, 
					Jerk						:= fJerk, 
					BufferMode					:= eBufferMode, 
					Options						:= , 
					Done						=> Out.Done, 
					Busy						=> Out.Busy, 
					Active						=> Out.Active, 
					CommandAborted				=> Out.CommandAborted, 
					Error						=> Out.Error, 
					ErrorID						=> Out.ErrorID);
	
pAbsolute2 										REF= Out;
pOut											REF= Out;

MoveAbsoluteEx2									:= TRUE;
END_METHOD

METHOD MoveModulo 								: REFERENCE TO Tc2_MC2.ST_McOutputs
VAR_INPUT
	bExecute									: BOOL;
END_VAR
IF bExecute THEN
	MoveModuloEx();
ELSE
	MoveModuloClear();
END_IF

MoveModulo										REF= pModulo;
END_METHOD

METHOD MoveModulo2 								: REFERENCE TO Tc2_MC2.ST_McOutputs
VAR_INPUT
	bExecute									: BOOL;
END_VAR
IF bExecute THEN
	MoveModuloEx2();
ELSE
	MoveModuloClear2();
END_IF

MoveModulo2										REF= pModulo2;
END_METHOD

METHOD MoveModuloClear 							: BOOL
VAR
	{attribute 'hide'}
	Out											: Tc2_MC2.ST_McOutputs;
END_VAR
mcMoveModulo(		Axis						:= Axis, 
					Execute						:= FALSE, 
					Done						=> Out.Done, 
					Busy						=> Out.Busy, 
					Active						=> Out.Active, 
					CommandAborted				=> Out.CommandAborted, 
					Error						=> Out.Error, 
					ErrorID						=> Out.ErrorID);
	
pModulo 										REF= Out;
pOut											REF= Out;

MoveModuloClear									:= TRUE;
END_METHOD

METHOD MoveModuloClear2 						: BOOL
VAR
	{attribute 'hide'}
	Out											: Tc2_MC2.ST_McOutputs;
END_VAR
mcMoveModulo2(		Axis						:= Axis, 
					Execute						:= FALSE, 
					Done						=> Out.Done, 
					Busy						=> Out.Busy, 
					Active						=> Out.Active, 
					CommandAborted				=> Out.CommandAborted, 
					Error						=> Out.Error, 
					ErrorID						=> Out.ErrorID);
	
pModulo2 										REF= Out;
pOut											REF= Out;

MoveModuloClear2								:= TRUE;
END_METHOD

METHOD MoveModuloCurrent 						: REFERENCE TO Tc2_MC2.ST_McOutputs
VAR_INPUT
	bExecute									: BOOL;
END_VAR
eDirection										:= Tc2_MC2.MC_Direction.MC_Current_Direction;

MoveModulo(bExecute := bExecute);

MoveModuloCurrent								REF= pModulo;
END_METHOD

METHOD MoveModuloCurrent2 						: REFERENCE TO Tc2_MC2.ST_McOutputs
VAR_INPUT
	bExecute									: BOOL;
END_VAR
eDirection										:= Tc2_MC2.MC_Direction.MC_Current_Direction;

MoveModulo(bExecute := bExecute);

MoveModuloCurrent2								REF= pModulo2;
END_METHOD

METHOD MoveModuloEx 							: BOOL
VAR
	{attribute 'hide'}
	Out											: Tc2_MC2.ST_McOutputs;
END_VAR
mcMoveModulo(		Axis						:= Axis, 
					Execute						:= TRUE, 
					Position					:= fPosition, 
					Velocity					:= fVelocity, 
					Acceleration				:= fAcceleration, 
					Deceleration				:= fDeceleration, 
					Jerk						:= fJerk,
					Direction					:= eDirection,
					BufferMode					:= eBufferMode, 
					Options						:= , 
					Done						=> Out.Done, 
					Busy						=> Out.Busy, 
					Active						=> Out.Active, 
					CommandAborted				=> Out.CommandAborted, 
					Error						=> Out.Error, 
					ErrorID						=> Out.ErrorID);
	
pModulo 										REF= Out;
pOut											REF= Out;

MoveModuloEx									:= TRUE;
END_METHOD

METHOD MoveModuloEx2 							: BOOL
VAR
	{attribute 'hide'}
	Out											: Tc2_MC2.ST_McOutputs;
END_VAR
mcMoveModulo2(		Axis						:= Axis, 
					Execute						:= TRUE, 
					Position					:= fPosition, 
					Velocity					:= fVelocity, 
					Acceleration				:= fAcceleration, 
					Deceleration				:= fDeceleration, 
					Jerk						:= fJerk,
					Direction					:= eDirection,
					BufferMode					:= eBufferMode, 
					Options						:= , 
					Done						=> Out.Done, 
					Busy						=> Out.Busy, 
					Active						=> Out.Active, 
					CommandAborted				=> Out.CommandAborted, 
					Error						=> Out.Error, 
					ErrorID						=> Out.ErrorID);
	
pModulo2 										REF= Out;
pOut											REF= Out;

MoveModuloEx2									:= TRUE;
END_METHOD

METHOD MoveModuloNeg 							: REFERENCE TO Tc2_MC2.ST_McOutputs
VAR_INPUT
	bExecute									: BOOL;
END_VAR
eDirection										:= Tc2_MC2.MC_Direction.MC_Negative_Direction;

MoveModulo(bExecute := bExecute);

MoveModuloNeg									REF= pModulo;
END_METHOD

METHOD MoveModuloNeg2 							: REFERENCE TO Tc2_MC2.ST_McOutputs
VAR_INPUT
	bExecute									: BOOL;
END_VAR
eDirection										:= Tc2_MC2.MC_Direction.MC_Negative_Direction;

MoveModulo(bExecute := bExecute);

MoveModuloNeg2									REF= pModulo2;
END_METHOD

METHOD MoveModuloPos 							: REFERENCE TO Tc2_MC2.ST_McOutputs
VAR_INPUT
	bExecute									: BOOL;
END_VAR
eDirection										:= Tc2_MC2.MC_Direction.MC_Positive_Direction;

MoveModulo(bExecute := bExecute);

MoveModuloPos									REF= pModulo;
END_METHOD

METHOD MoveModuloPos2 							: REFERENCE TO Tc2_MC2.ST_McOutputs
VAR_INPUT
	bExecute									: BOOL;
END_VAR
eDirection										:= Tc2_MC2.MC_Direction.MC_Positive_Direction;

MoveModulo(bExecute := bExecute);

MoveModuloPos2									REF= pModulo2;
END_METHOD

METHOD MoveModuloShort 							: REFERENCE TO Tc2_MC2.ST_McOutputs
VAR_INPUT
	bExecute									: BOOL;
END_VAR
eDirection										:= Tc2_MC2.MC_Direction.MC_Shortest_Way;

MoveModulo(bExecute := bExecute);

MoveModuloShort									REF= pModulo;
END_METHOD

METHOD MoveModuloShort2 						: REFERENCE TO Tc2_MC2.ST_McOutputs
VAR_INPUT
	bExecute									: BOOL;
END_VAR
eDirection										:= Tc2_MC2.MC_Direction.MC_Shortest_Way;

MoveModulo(bExecute := bExecute);

MoveModuloShort2								REF= pModulo2;
END_METHOD

METHOD MoveRelative 							: REFERENCE TO Tc2_MC2.ST_McOutputs
VAR_INPUT
	bExecute									: BOOL;
END_VAR
IF bExecute THEN
	MoveRelativeEx();
//	Out		:= MoveRelativeEx.Out;
ELSE
	MoveRelativeClear();
END_IF

MoveRelative									REF= pRelative;
END_METHOD

METHOD MoveRelative2 							: REFERENCE TO Tc2_MC2.ST_McOutputs
VAR_INPUT
	bExecute									: BOOL;
END_VAR
IF bExecute THEN
	MoveRelativeEx2();
ELSE
	MoveRelativeClear2();
END_IF

MoveRelative2									REF= pRelative2;
END_METHOD

METHOD MoveRelativeClear 						: BOOL
VAR
	{attribute 'hide'}
	Out											: Tc2_MC2.ST_McOutputs;
END_VAR
mcMoveRelative(		Axis						:= Axis, 
					Execute						:= FALSE, 
					Done						=> Out.Done, 
					Busy						=> Out.Busy, 
					Active						=> Out.Active, 
					CommandAborted				=> Out.CommandAborted, 
					Error						=> Out.Error, 
					ErrorID						=> Out.ErrorID);
	
pRelative 										REF= Out;
pOut											REF= Out;

MoveRelativeClear								:= TRUE;
END_METHOD

METHOD MoveRelativeClear2 						: BOOL
VAR
	{attribute 'hide'}
	Out											: Tc2_MC2.ST_McOutputs;
END_VAR
mcMoveRelative2(	Axis						:= Axis, 
					Execute						:= FALSE, 
					Done						=> Out.Done, 
					Busy						=> Out.Busy, 
					Active						=> Out.Active, 
					CommandAborted				=> Out.CommandAborted, 
					Error						=> Out.Error, 
					ErrorID						=> Out.ErrorID);
	
pRelative2 										REF= Out;
pOut											REF= Out;

MoveRelativeClear2								:= TRUE;
END_METHOD

METHOD MoveRelativeEx 							: BOOL

VAR
	{attribute 'hide'}
	Out											: Tc2_MC2.ST_McOutputs;
END_VAR
mcMoveRelative(		Axis						:= Axis, 
					Execute						:= TRUE, 
					Distance					:= fDistance, 
					Velocity					:= fVelocity, 
					Acceleration				:= fAcceleration, 
					Deceleration				:= fDeceleration, 
					Jerk						:= fJerk, 
					BufferMode					:= eBufferMode, 
					Options						:= , 
					Done						=> Out.Done, 
					Busy						=> Out.Busy, 
					Active						=> Out.Active, 
					CommandAborted				=> Out.CommandAborted, 
					Error						=> Out.Error, 
					ErrorID						=> Out.ErrorID);
	
pRelative 										REF= Out;
pOut											REF= Out;

MoveRelativeEx									:= TRUE;
END_METHOD

METHOD MoveRelativeEx2 							: BOOL
VAR
	{attribute 'hide'}
	Out											: Tc2_MC2.ST_McOutputs;
END_VAR
mcMoveRelative2(	Axis						:= Axis, 
					Execute						:= TRUE, 
					Distance					:= fDistance, 
					Velocity					:= fVelocity, 
					Acceleration				:= fAcceleration, 
					Deceleration				:= fDeceleration, 
					Jerk						:= fJerk, 
					BufferMode					:= eBufferMode, 
					Options						:= , 
					Done						=> Out.Done, 
					Busy						=> Out.Busy, 
					Active						=> Out.Active, 
					CommandAborted				=> Out.CommandAborted, 
					Error						=> Out.Error, 
					ErrorID						=> Out.ErrorID);
	
pRelative2 										REF= Out;
pOut											REF= Out;

MoveRelativeEx2									:= TRUE;
END_METHOD

METHOD MoveVelocity 							: REFERENCE TO Tc2_MC2.ST_McOutputs
VAR_INPUT
	bExecute									: BOOL;
END_VAR
IF bExecute THEN
	MoveVelocityEx();
ELSE
	MoveVelocityClear();
END_IF

MoveVelocity									REF= pVelocity;
END_METHOD

METHOD MoveVelocity2 							: REFERENCE TO Tc2_MC2.ST_McOutputs
VAR_INPUT
	bExecute									: BOOL;
END_VAR
IF bExecute THEN
	MoveVelocityEx2();
ELSE
	MoveVelocityClear2();
END_IF

MoveVelocity2									REF= pVelocity2;
END_METHOD

METHOD MoveVelocityClear 						: BOOL
VAR
	{attribute 'hide'}
	Out											: Tc2_MC2.ST_McOutputs;
END_VAR
mcMoveVelocity(		Axis						:= Axis, 
					Execute						:= FALSE, 
					InVelocity					=> Out.Done, 
					Busy						=> Out.Busy, 
					Active						=> Out.Active, 
					CommandAborted				=> Out.CommandAborted, 
					Error						=> Out.Error, 
					ErrorID						=> Out.ErrorID);

pVelocity 										REF= Out;
pOut											REF= Out;

MoveVelocityClear								:= TRUE;
END_METHOD

METHOD MoveVelocityClear2 						: BOOL
VAR
	{attribute 'hide'}
	Out											: Tc2_MC2.ST_McOutputs;
END_VAR
mcMoveVelocity2(	Axis						:= Axis, 
					Execute						:= FALSE, 
					InVelocity					=> Out.Done, 
					Busy						=> Out.Busy, 
					Active						=> Out.Active, 
					CommandAborted				=> Out.CommandAborted, 
					Error						=> Out.Error, 
					ErrorID						=> Out.ErrorID);

pVelocity2 										REF= Out;
pOut											REF= Out;

MoveVelocityClear2								:= TRUE;
END_METHOD

METHOD MoveVelocityEx 							: BOOL
VAR
	{attribute 'hide'}
	Out											: Tc2_MC2.ST_McOutputs;
END_VAR
mcMoveVelocity(		Axis						:= Axis, 
					Execute						:= TRUE, 
					Velocity					:= fVelocity, 
					Acceleration				:= fAcceleration, 
					Deceleration				:= fDeceleration, 
					Jerk						:= fJerk, 
					Direction					:= eDirection, 
					BufferMode					:= eBufferMode, 
					Options						:= , 
					InVelocity					=> Out.Done, 
					Busy						=> Out.Busy, 
					Active						=> Out.Active, 
					CommandAborted				=> Out.CommandAborted, 
					Error						=> Out.Error, 
					ErrorID						=> Out.ErrorID);

pVelocity 										REF= Out;
pOut											REF= Out;

MoveVelocityEx									:= TRUE;
END_METHOD

METHOD MoveVelocityEx2 							: BOOL
VAR
	{attribute 'hide'}
	Out											: Tc2_MC2.ST_McOutputs;
END_VAR
mcMoveVelocity2(	Axis						:= Axis, 
					Execute						:= TRUE, 
					Velocity					:= fVelocity, 
					Acceleration				:= fAcceleration, 
					Deceleration				:= fDeceleration, 
					Jerk						:= fJerk, 
					Direction					:= eDirection, 
					BufferMode					:= eBufferMode, 
					Options						:= , 
					InVelocity					=> Out.Done, 
					Busy						=> Out.Busy, 
					Active						=> Out.Active, 
					CommandAborted				=> Out.CommandAborted, 
					Error						=> Out.Error, 
					ErrorID						=> Out.ErrorID);

pVelocity2 										REF= Out;
pOut											REF= Out;

MoveVelocityEx2									:= TRUE;
END_METHOD

METHOD MoveVelocityNegative 					: REFERENCE TO Tc2_MC2.ST_McOutputs
VAR_INPUT
	bExecute									: BOOL;
END_VAR
eDirection										:= Tc2_MC2.MC_Direction.MC_Negative_Direction;
MoveVelocity(bExecute := bExecute);

MoveVelocityNegative							REF= pVelocity;
END_METHOD

METHOD MoveVelocityNegative2 					: REFERENCE TO Tc2_MC2.ST_McOutputs
VAR_INPUT
	bExecute									: BOOL;
END_VAR
eDirection										:= Tc2_MC2.MC_Direction.MC_Negative_Direction;
MoveVelocity2(bExecute := bExecute);

MoveVelocityNegative2							REF= pVelocity;
END_METHOD

METHOD MoveVelocityNegativeDyn 					: REFERENCE TO Tc2_MC2.ST_McOutputs
VAR_INPUT
	bExecute									: BOOL;
END_VAR
;
END_METHOD

METHOD MoveVelocityPositive 					: REFERENCE TO Tc2_MC2.ST_McOutputs
VAR_INPUT
	bExecute									: BOOL;
END_VAR
eDirection										:= Tc2_MC2.MC_Direction.MC_Positive_Direction;
MoveVelocity(bExecute := bExecute);

MoveVelocityPositive							REF= pVelocity;
END_METHOD

METHOD MoveVelocityPositive2 					: REFERENCE TO Tc2_MC2.ST_McOutputs
VAR_INPUT
	bExecute									: BOOL;
END_VAR
eDirection										:= Tc2_MC2.MC_Direction.MC_Positive_Direction;
MoveVelocity2(bExecute := bExecute);

MoveVelocityPositive2							REF= pVelocity2;
END_METHOD

METHOD MoveVelocityPositiveDyn 					: REFERENCE TO Tc2_MC2.ST_McOutputs
VAR_INPUT
	bEnable										: BOOL;
END_VAR
VAR_INST
	{attribute 'hide'}
	fVelocityOld								: LREAL;
	{attribute 'hide'}
	Out1										: Tc2_MC2.ST_McOutputs;
	{attribute 'hide'}
	Out2										: Tc2_MC2.ST_McOutputs;
	{attribute 'hide'}
	bExecute1									: BOOL;
	{attribute 'hide'}
	bExecute2									: BOOL;
END_VAR
IF bEnable THEN
	eBufferMode									:= Tc2_MC2.MC_BufferMode.MC_Aborting;
	IF fVelocity <> fVelocityOld THEN
		IF NOT Out1.Active THEN
			bExecute1 							:= TRUE;
			bExecute2 							:= FALSE;
		ELSE
			bExecute1 							:= FALSE;
			bExecute2 							:= TRUE;
		END_IF
		fVelocityOld := fVelocity;
	END_IF
END_IF

Out1 											:= MoveVelocityPositive(bExecute := bExecute1);
Out2 											:= MoveVelocityPositive2(bExecute := bExecute2);
END_METHOD

{attribute 'monitoring' := 'variable'}
PROPERTY nErrorId 								: UDINT
GET
nErrorId											:= Axis.Status.ErrorID;
END_GET
END_PROPERTY

{attribute 'monitoring' := 'variable'}
PROPERTY nErrorIdFiltered 								: UDINT
GET
nErrorIdFiltered								:= SEL(bConsequentialError,Axis.Status.ErrorID,0);
END_GET
END_PROPERTY

{attribute 'monitoring' := 'variable'}
PROPERTY pAbsolute 								: REFERENCE TO Tc2_MC2.ST_McOutputs
GET
pAbsolute										REF= _stAbsolute;
END_GET
SET
_stAbsolute										:= pAbsolute;
END_SET
END_PROPERTY

{attribute 'monitoring' := 'variable'}
PROPERTY pAbsolute2 							: REFERENCE TO Tc2_MC2.ST_McOutputs
GET
pAbsolute2										REF= _stAbsolute2;
END_GET
SET
_stAbsolute2									:= pAbsolute2;
END_SET
END_PROPERTY

{attribute 'monitoring' := 'variable'}
PROPERTY pEStop 								: REFERENCE TO Tc2_MC2.ST_McOutputs
GET
pEStop											REF= _stEStop;
END_GET
SET
_stEStop										:= pEStop;
END_SET
END_PROPERTY

{attribute 'monitoring' := 'variable'}
PROPERTY pGear 									: REFERENCE TO Tc2_MC2.ST_McOutputs
GET
pGear											REF= _stGear;
END_GET
SET
_stGear											:= pGear;
END_SET
END_PROPERTY

{attribute 'monitoring' := 'variable'}
PROPERTY pHalt 									: REFERENCE TO Tc2_MC2.ST_McOutputs
GET
pHalt											REF= _stHalt;
END_GET
SET
_stHalt											:= pHalt;
END_SET
END_PROPERTY

{attribute 'monitoring' := 'variable'}
PROPERTY pHome 									: REFERENCE TO Tc2_MC2.ST_McOutputs
GET
pHome											REF= _stHome;
END_GET
SET
_stHome											:= pHome;
END_SET
END_PROPERTY

{attribute 'monitoring' := 'variable'}
PROPERTY pJog 									: REFERENCE TO Tc2_MC2.ST_McOutputs
GET
pJog											REF= _stJog;
END_GET
SET
_stJog											:= pJog;
END_SET
END_PROPERTY

{attribute 'monitoring' := 'variable'}
PROPERTY pLimitSwitch 							: REFERENCE TO Tc2_MC2.ST_McOutputs
GET
pLimitSwitch								REF= _stLimitSwitch;
END_GET
SET
_stLimitSwitch									:= pLimitSwitch;
END_SET
END_PROPERTY

{attribute 'monitoring' := 'variable'}
PROPERTY pModulo 								: REFERENCE TO Tc2_MC2.ST_McOutputs
GET
pModulo											REF= _stModulo;
END_GET
SET
_stModulo										:= pModulo;
END_SET
END_PROPERTY

{attribute 'monitoring' := 'variable'}
PROPERTY pModulo2 								: REFERENCE TO Tc2_MC2.ST_McOutputs
GET
pModulo2										REF= _stModulo2;
END_GET
SET
_stModulo2										:= pModulo2;
END_SET
END_PROPERTY

{attribute 'monitoring' := 'variable'}
// Only motion FBs
PROPERTY pOut 									: REFERENCE TO Tc2_MC2.ST_McOutputs
GET
pOut											REF= _stOut;
END_GET
SET
_stOut											:= pOut;
END_SET
END_PROPERTY

METHOD Power 									: REFERENCE TO Tc2_MC2.ST_McOutputs
// SS1 read status
IF bEnable AND NOT pEStop.Done THEN
	Enable();
ELSE
	Disable();
END_IF

Power											REF= pPower;
END_METHOD

{attribute 'monitoring' := 'variable'}
PROPERTY pPower 								: REFERENCE TO Tc2_MC2.ST_McOutputs
GET
pPower											REF= _stPower;
END_GET
SET
_stPower										:= pPower;
END_SET
END_PROPERTY

{attribute 'monitoring' := 'variable'}
PROPERTY pRelative 								: REFERENCE TO Tc2_MC2.ST_McOutputs
GET
pRelative										REF= _stRelative;
END_GET
SET
_stRelative										:= pRelative;
END_SET
END_PROPERTY

{attribute 'monitoring' := 'variable'}
PROPERTY pRelative2 							: REFERENCE TO Tc2_MC2.ST_McOutputs
GET
pRelative2										REF= _stRelative2;
END_GET
SET
_stRelative2									:= pRelative2;
END_SET
END_PROPERTY

{attribute 'monitoring' := 'variable'}
PROPERTY pReset 								: REFERENCE TO Tc2_MC2.ST_McOutputs
GET
pReset											REF= _stReset;
END_GET
SET
_stReset										:= pReset;
END_SET
END_PROPERTY

PROPERTY pSetPos 								: REFERENCE TO Tc2_MC2.ST_McOutputs
GET
pSetPos											REF= _stSetPos;
END_GET
SET
_stSetPos										:= pSetPos;
END_SET
END_PROPERTY

{attribute 'monitoring' := 'variable'}
PROPERTY pStop 									: REFERENCE TO Tc2_MC2.ST_McOutputs
GET
pStop											REF= _stStop;
END_GET
SET
_stStop											:= pStop;
END_SET
END_PROPERTY

{attribute 'monitoring' := 'variable'}
PROPERTY pSuperimposed 						: REFERENCE TO Tc2_MC2.ST_McOutputs
GET
pSuperimposed									REF= _stSuperimposed;
END_GET
SET
_stSuperimposed									:= pSuperimposed;
END_SET
END_PROPERTY

{attribute 'monitoring' := 'variable'}
PROPERTY pVelocity 								: REFERENCE TO Tc2_MC2.ST_McOutputs
GET
pVelocity										REF= _stVelocity;
END_GET
SET
_stVelocity										:= pVelocity;
END_SET
END_PROPERTY

{attribute 'monitoring' := 'variable'}
PROPERTY pVelocity2 							: REFERENCE TO Tc2_MC2.ST_McOutputs
GET
pVelocity2										REF= _stVelocity2;
END_GET
SET
_stVelocity2									:= pVelocity2;
END_SET
END_PROPERTY

METHOD PRIVATE ReadParameterSet 				: REFERENCE TO Tc2_MC2.ST_McOutputs
VAR_INPUT
	bExecute									: BOOL;
END_VAR
VAR_INST
	bAxisParametersError						: BOOL;
	{attribute 'hide'}
	mcReadParameterSet							: Tc2_MC2.MC_ReadParameterSet;
END_VAR
VAR
	{attribute 'hide'}
	Out											: Tc2_MC2.ST_McOutputs;
END_VAR
mcReadParameterSet(	Parameter					:= stParameters,
					Axis						:= Axis,
					Execute						:= bExecute,
					Done						=> Out.Done,
					Busy						=> Out.Busy,
					Error						=> Out.Error,
					ErrorID						=> Out.ErrorID);
					
ReadParameterSet								REF= Out;
END_METHOD

METHOD Reset 									: REFERENCE TO Tc2_MC2.ST_McOutputs
VAR_INPUT
	bExecute									: BOOL;
END_VAR
IF bExecute THEN
	ResetEx();
ELSE
	ResetClear();
END_IF

Reset											REF= pReset;
END_METHOD

METHOD ResetClear 								: BOOL
VAR
	{attribute 'hide'}
	Out											: Tc2_MC2.ST_McOutputs;
END_VAR
mcReset(			Axis						:= Axis, 
					Execute						:= FALSE, 
					Done						=> Out.Done, 
					Busy						=> Out.Busy, 
					Error						=> Out.Error, 
					ErrorID						=> Out.ErrorID);
	
pReset 											REF= Out;

ResetClear										:= TRUE;
END_METHOD

METHOD ResetEx 									: BOOL
VAR
	{attribute 'hide'}
	Out											: Tc2_MC2.ST_McOutputs;
END_VAR
mcReset(			Axis						:= Axis, 
					Execute						:= TRUE, 
					Done						=> Out.Done, 
					Busy						=> Out.Busy, 
					Error						=> Out.Error, 
					ErrorID						=> Out.ErrorID);
	
pReset 											REF= Out;

ResetEx											:= TRUE;
END_METHOD

METHOD SetPos 									: REFERENCE TO Tc2_MC2.ST_McOutputs
VAR_INPUT
	bExecute									: BOOL;
	bMode										: BOOL;	// RELATIVE=True, ABSOLUTE=False (Default)
	stOptions									: Tc2_MC2.ST_SetPositionOptions;
END_VAR
IF bExecute THEN
	SetPosEx(bMode := bMode, stOptions := stOptions);
ELSE
	SetPosClear();
END_IF

SetPos											REF= pSetPos;
END_METHOD

METHOD SetPosAbs0ClearLag 						: REFERENCE TO Tc2_MC2.ST_McOutputs
VAR_INPUT
	bExecute									: BOOL;
END_VAR
VAR
	{attribute 'hide'}
	stOptions									: Tc2_MC2.ST_SetPositionOptions;	
END_VAR
stOptions.ClearPositionLag						:= TRUE;
fPosition										:= 0.0;

SetPos(bExecute := bExecute, bMode := FALSE, stOptions := stOptions);

SetPosAbs0ClearLag								REF= pSetPos;
END_METHOD

METHOD SetPosAbsClearLag 						: REFERENCE TO Tc2_MC2.ST_McOutputs
VAR_INPUT
	bExecute									: BOOL;
END_VAR
VAR
	{attribute 'hide'}
	stOptions									: Tc2_MC2.ST_SetPositionOptions;	
END_VAR
stOptions.ClearPositionLag						:= TRUE;

SetPos(bExecute := bExecute, bMode := FALSE, stOptions := stOptions);

SetPosAbsClearLag								REF= pSetPos;
END_METHOD

METHOD SetPosClear 								: BOOL
VAR
	{attribute 'hide'}
	Out											: Tc2_MC2.ST_McOutputs;
END_VAR
mcSetPos(			Axis						:= Axis, 
					Execute						:= FALSE, 
					Done						=> Out.Done, 
					Busy						=> Out.Busy, 
					Error						=> Out.Error, 
					ErrorID						=> Out.ErrorID);
					
pSetPos 										REF= Out;

SetPosClear										:= TRUE;
END_METHOD

METHOD SetPosEx 								: BOOL
VAR_INPUT
	bMode										: BOOL;	// RELATIVE=True, ABSOLUTE=False (Default)
	stOptions									: Tc2_MC2.ST_SetPositionOptions;
END_VAR
VAR
	{attribute 'hide'}
	Out											: Tc2_MC2.ST_McOutputs;
END_VAR
mcSetPos(			Axis						:= Axis, 
					Execute						:= TRUE, 
					Position					:= fPosition, 
					Mode						:= bMode, 
					Options						:= stOptions, 
					Done						=> Out.Done, 
					Busy						=> Out.Busy, 
					Error						=> Out.Error, 
					ErrorID						=> Out.ErrorID);
					
pSetPos 										REF= Out;

SetPosEx										:= TRUE;
END_METHOD

METHOD SetPosRelClearLag 						: REFERENCE TO Tc2_MC2.ST_McOutputs
VAR_INPUT
	bExecute									: BOOL;
END_VAR
VAR
	{attribute 'hide'}
	stOptions									: Tc2_MC2.ST_SetPositionOptions;	
END_VAR
stOptions.ClearPositionLag						:= TRUE;

SetPos(bExecute := bExecute, bMode := TRUE, stOptions := stOptions);

SetPosRelClearLag								REF= pSetPos;
END_METHOD

PROPERTY stAxisStatus: reference to ST_AxisStatus;
GET
stAxisStatus ref= Axis.Status;
END_GET
END_PROPERTY

METHOD Stop 									: REFERENCE TO Tc2_MC2.ST_McOutputs
VAR_INPUT
	bExecute									: BOOL;
END_VAR
IF bExecute THEN
	StopEx();
ELSE
	StopClear();
END_IF

Stop											REF= pStop;
END_METHOD

METHOD StopClear 								: BOOL
VAR
	{attribute 'hide'}
	Out											: Tc2_MC2.ST_McOutputs;
END_VAR
mcStop(				Axis						:= Axis, 
					Execute						:= FALSE, 
					Done						=> Out.Done, 
					Busy						=> Out.Busy, 
					Active						=> Out.Active, 
					CommandAborted				=> Out.CommandAborted, 
//					Error						=> Out.Error, 
					ErrorID						=> Out.ErrorID);
Out.Error	:= FALSE;

pStop				 							REF= Out;

StopClear										:= TRUE;
END_METHOD

METHOD StopEx 									: BOOL
VAR
	{attribute 'hide'}
	Out											: Tc2_MC2.ST_McOutputs;
END_VAR
mcStop(				Axis						:= Axis, 
					Execute						:= TRUE, 
					Deceleration				:= fDeceleration, 
					Jerk						:= fJerk, 
					Options						:= , 
					Done						=> Out.Done, 
					Busy						=> Out.Busy, 
					Active						=> Out.Active, 
					CommandAborted				=> Out.CommandAborted, 
					Error						=> Out.Error, 
					ErrorID						=> Out.ErrorID);

pStop				 							REF= Out;

StopEx											:= TRUE;
END_METHOD

END_FUNCTION_BLOCK

// ---- POUs/FB/AxisControl/Internal/FB_NcSWLimitSwitchCtrlv2.TcPOU
//==================================================================================================
//							Beckhoff Automation Poland
//									03.01.2023
//
// Code owner: TG
//
// Sample code to maitenance software limit switches
//
// Used libraries: 
//	Tc2_MC2							|| 3.3.48.0
//	Tc2_System						|| 3.4.26.0
//
//
// 	v2.0 	|| TC v 3.1.4024.35 	|| Second edition - OOP based
// 	v1.0 	|| TC v 3.1.4020.32 	|| First edition
//==================================================================================================
{attribute 'reflection'}
FUNCTION_BLOCK FB_NcSWLimitSwitchCtrlv2
VAR CONSTANT
	udiIDXGRP_OFFS								: UDINT := 16#0000_5000;
END_VAR
VAR
	{attribute 'instance-path'}
	{attribute 'noinit'}
	sInstancePath								: STRING;

	_stRead										: Tc2_MC2.ST_McOutputs;
	_stWrite									: Tc2_MC2.ST_McOutputs;
	_lrLimitSwitchPositionMin					: LREAL 		:= 0;
	_lrLimitSwitchPositionMax					: LREAL 		:= 0;
	_bLimitSwitchStateMin						: BOOL 			:= FALSE;
	_bLimitSwitchStateMax						: BOOL 			:= FALSE;
	bAxisIdError								: BOOL;
END_VAR

PROPERTY LimitSwitchPositionMax 				: LREAL
GET
LimitSwitchPositionMax							:= _lrLimitSwitchPositionMax;
END_GET
SET
_lrLimitSwitchPositionMax						:= LimitSwitchPositionMax;
END_SET
END_PROPERTY

PROPERTY LimitSwitchPositionMin 				: LREAL
GET
LimitSwitchPositionMin							:= _lrLimitSwitchPositionMin;
END_GET
SET
_lrLimitSwitchPositionMin						:= LimitSwitchPositionMin;
END_SET
END_PROPERTY

PROPERTY LimitSwitchStateMax 					: BOOL
GET
LimitSwitchStateMax								:= _bLimitSwitchStateMax;
END_GET
SET
_bLimitSwitchStateMax							:= LimitSwitchStateMax;
END_SET
END_PROPERTY

PROPERTY LimitSwitchStateMin 					: BOOL
GET
LimitSwitchStateMin							:= _bLimitSwitchStateMin;
END_GET
SET
_bLimitSwitchStateMin							:= LimitSwitchStateMin;
END_SET
END_PROPERTY

PROPERTY pRead 							: Tc2_MC2.ST_McOutputs
GET
pRead											:= _stRead;
END_GET
SET
_stRead											:= pRead;
END_SET
END_PROPERTY

PROPERTY pWrite 							: Tc2_MC2.ST_McOutputs
GET
pWrite											:= _stWrite;
END_GET
SET
_stWrite										:= pWrite;
END_SET
END_PROPERTY

// Needs one cycle extra with false execution, after busy false
METHOD ReadBool 								: Tc2_MC2.ST_McOutputs
VAR_INPUT
	bExecute									: BOOL;
	nAxisID										: UDINT;
	nOffset										: UDINT;
END_VAR
VAR_OUTPUT
	bOut										: BOOL;
END_VAR
VAR_INST
	fbADSREAD									: ADSREAD;
	wData										: WORD;
	nStep										: DINT;
END_VAR
VAR
	Out											: Tc2_MC2.ST_McOutputs;
	Message										: STRING;
END_VAR
IF nAxisID = 0 THEN
	
	IF NOT bAxisIdError THEN
		ADSLOGSTR(ADSLOG_MSGTYPE_ERROR,'FB_NcSWLimitSwitchCtrl critical error - Axis ID not assigned! FB instance: %s',sInstancePath);
	END_IF
	
	bAxisIdError 								:= TRUE;
	RETURN;	
END_IF

